# B&R Automation Studio project TD52 (part 51)

#### c_clutch_CANCyclic.st - Init, cyclic, exit code
```iecst
(*******************************************************************************
NOxSensor: 	 		CAN communication to Horton CAN bus device (cyclic)

This code is confidential and proprietary to the INNIO Company.
It may not be used in any form, or reproduced in any manner, without the express
written permission of the INNIO Company.
Copyright, INNIO Company, 2026

Customized modifications: -
------------------------

History:
-------

V4.16.00.00	06.01.2026	Bencze,  HORTON CAN bus device Cyclic code

Instructions for use:
--------------------

-----------------------------------------------------------------------------------------------------------------------------------------------	*)

PROGRAM _CYCLIC

	// Trigger reception of the data
	TON_1sTick(IN := NOT TON_1sTick.Q, PT := T#800ms);				(* 80ms + 2 times cycle time = 100ms *)

	// CAN communication timeout warning timers
	FOR DeviceNumber := 0 TO 3 DO
		TON_10sTick_DumpRadiator[DeviceNumber](IN := NOT DumpRadiator_PGN_Message_CS1[DeviceNumber].CommandDone OR NOT DumpRadiator_PGN_Message_CS2[DeviceNumber].CommandDone, PT := T#9800ms);
		TON_10sTick_AirInFan[DeviceNumber](IN := NOT AirInFan_PGN_Message_CS1[DeviceNumber].CommandDone OR NOT AirInFan_PGN_Message_CS2[DeviceNumber].CommandDone, PT := T#9800ms);
	END_FOR;

	// DumpRadiator - Connection with Map Services
	DumpRadiator_PGN_Message_CS1[0].MpLink := ADR(Dump_Radiator_1_CS1);
	DumpRadiator_PGN_Message_CS2[0].MpLink := ADR(Dump_Radiator_1_CS2);
	DumpRadiator_PGN_Message_CS1[1].MpLink := ADR(Dump_Radiator_2_CS1);
	DumpRadiator_PGN_Message_CS2[1].MpLink := ADR(Dump_Radiator_2_CS2);
	DumpRadiator_PGN_Message_CS1[2].MpLink := ADR(Dump_Radiator_3_CS1);
	DumpRadiator_PGN_Message_CS2[2].MpLink := ADR(Dump_Radiator_3_CS2);
	DumpRadiator_PGN_Message_CS1[3].MpLink := ADR(Dump_Radiator_4_CS1);
	DumpRadiator_PGN_Message_CS2[3].MpLink := ADR(Dump_Radiator_4_CS2);

	// AirInFan - Connection with Map Services
	AirInFan_PGN_Message_CS1[0].MpLink := ADR(Air_Inlet_Fan_1_CS1);
	AirInFan_PGN_Message_CS2[0].MpLink := ADR(Air_Inlet_Fan_1_CS2);
	AirInFan_PGN_Message_CS1[1].MpLink := ADR(Air_Inlet_Fan_2_CS1);
	AirInFan_PGN_Message_CS2[1].MpLink := ADR(Air_Inlet_Fan_2_CS2);
	AirInFan_PGN_Message_CS1[2].MpLink := ADR(Air_Inlet_Fan_3_CS1);
	AirInFan_PGN_Message_CS2[2].MpLink := ADR(Air_Inlet_Fan_3_CS2);
	AirInFan_PGN_Message_CS1[3].MpLink := ADR(Air_Inlet_Fan_4_CS1);
	AirInFan_PGN_Message_CS2[3].MpLink := ADR(Air_Inlet_Fan_4_CS2);

	FOR DeviceNumber := 0 TO 3 DO
		// Specific messages 1 (CS1 - Horton documentation)
		DumpRadiator_PGN_Message_CS1[DeviceNumber].Enable := TRUE;
		DumpRadiator_PGN_Message_CS1[DeviceNumber].Receive := TON_1sTick.Q;
		DumpRadiator_PGN_Message_CS1[DeviceNumber].PGN := 65470;
		DumpRadiator_PGN_Message_CS1[DeviceNumber].Priority := 5;
		DumpRadiator_PGN_Message_CS1[DeviceNumber].DataLength := 8;
		DumpRadiator_PGN_Message_CS1[DeviceNumber].Data := ADR(DumpRadiator_CS1_RawData[DeviceNumber]);
		DumpRadiator_PGN_Message_CS1[DeviceNumber]();

		// Specific messages 2 (CS2 - Horton documentation)
		DumpRadiator_PGN_Message_CS2[DeviceNumber].Enable := TRUE;
		DumpRadiator_PGN_Message_CS2[DeviceNumber].Receive := TON_1sTick.Q;
		DumpRadiator_PGN_Message_CS2[DeviceNumber].PGN := 65469;
		DumpRadiator_PGN_Message_CS2[DeviceNumber].Priority := 5;
		DumpRadiator_PGN_Message_CS2[DeviceNumber].DataLength := 8;
		DumpRadiator_PGN_Message_CS2[DeviceNumber].Data := ADR(DumpRadiator_CS2_RawData[DeviceNumber]);
		DumpRadiator_PGN_Message_CS2[DeviceNumber]();

		// Specific messages 1 (CS1 - Horton documentation)
		AirInFan_PGN_Message_CS1[DeviceNumber].Enable := TRUE;
		AirInFan_PGN_Message_CS1[DeviceNumber].Receive := TON_1sTick.Q;
		AirInFan_PGN_Message_CS1[DeviceNumber].PGN := 65470;
		AirInFan_PGN_Message_CS1[DeviceNumber].Priority := 5;
		AirInFan_PGN_Message_CS1[DeviceNumber].DataLength := 8;
		AirInFan_PGN_Message_CS1[DeviceNumber].Data := ADR(AirInFan_CS1_RawData[DeviceNumber]);
		AirInFan_PGN_Message_CS1[DeviceNumber]();

		// Specific messages 2 (CS2 - Horton documentation)
		AirInFan_PGN_Message_CS2[DeviceNumber].Enable := TRUE;
		AirInFan_PGN_Message_CS2[DeviceNumber].Receive := TON_1sTick.Q;
		AirInFan_PGN_Message_CS2[DeviceNumber].PGN := 65469;
		AirInFan_PGN_Message_CS2[DeviceNumber].Priority := 5;
		AirInFan_PGN_Message_CS2[DeviceNumber].DataLength := 8;
		AirInFan_PGN_Message_CS2[DeviceNumber].Data := ADR(AirInFan_CS2_RawData[DeviceNumber]);
		AirInFan_PGN_Message_CS2[DeviceNumber]();
	END_FOR;

	FOR DeviceNumber := 0 TO 3 DO
		// DumpRadiator - Measured Fan Speed and Speed signal from PLC (AO)
		MM2VIS_ThisPlant.rDumpRadiator_Speed[DeviceNumber] := DumpRadiator_CS1_RawData[DeviceNumber].Data2 + DumpRadiator_CS1_RawData[DeviceNumber].Data3 * 256; // Fan speed to the device
		MM2VIS_ThisPlant.rDumpRadiator_InputSpeed[DeviceNumber] := DumpRadiator_CS1_RawData[DeviceNumber].Data6 + DumpRadiator_CS1_RawData[DeviceNumber].Data7 * 256; // Fan speed measurement coming to PLC

		// AirInFan - Measured Fan Speed and Speed signal from PLC (AO)
		MM2VIS_ThisPlant.rAirInFan_Speed[DeviceNumber] := AirInFan_CS1_RawData[DeviceNumber].Data2 + AirInFan_CS1_RawData[DeviceNumber].Data3 * 256; // Fan speed to the device
		MM2VIS_ThisPlant.rAirInFan_InputSpeed[DeviceNumber]  := AirInFan_CS1_RawData[DeviceNumber].Data6 + AirInFan_CS1_RawData[DeviceNumber].Data7 * 256; // Fan speed measurement coming to PLC
	END_FOR;

	// Dump Radiators are running
	MM2VIS_ThisPlant.bDumpRadiatorRUN[0] := (MM2VIS_ThisPlant.rDumpRadiator_InputSpeed[0] >= OUT_CU.rCust_SparePara[26]);
	MM2VIS_ThisPlant.bDumpRadiatorRUN[1] := (MM2VIS_ThisPlant.rDumpRadiator_InputSpeed[1] >= OUT_CU.rCust_SparePara[26]);
	MM2VIS_ThisPlant.bDumpRadiatorRUN[2] := (MM2VIS_ThisPlant.rDumpRadiator_InputSpeed[2] >= OUT_CU.rCust_SparePara[26]);
	MM2VIS_ThisPlant.bDumpRadiatorRUN[3] := (MM2VIS_ThisPlant.rDumpRadiator_InputSpeed[3] >= OUT_CU.rCust_SparePara[26]);
	// Air Inlet Fans are running
	MM2VIS_ThisPlant.bAirInFanRUN[0] := (MM2VIS_ThisPlant.rAirInFan_InputSpeed[0] >= OUT_CU.rCust_SparePara[39]);
	MM2VIS_ThisPlant.bAirInFanRUN[1] := (MM2VIS_ThisPlant.rAirInFan_InputSpeed[1] >= OUT_CU.rCust_SparePara[39]);
	MM2VIS_ThisPlant.bAirInFanRUN[2] := (MM2VIS_ThisPlant.rAirInFan_InputSpeed[2] >= OUT_CU.rCust_SparePara[39]);
	MM2VIS_ThisPlant.bAirInFanRUN[3] := (MM2VIS_ThisPlant.rAirInFan_InputSpeed[3] >= OUT_CU.rCust_SparePara[39]);

	FOR DeviceNumber := 0 TO 3 DO
		// DumpRadiator - Clutch status
		MM2VIS_ThisPlant.bDumpRadiator_FanCmdLThanMICS[DeviceNumber] := DumpRadiator_CS2_RawData[DeviceNumber].Data2.3; // Fan command less than MICS (Min Controllable Fan Speed)
		MM2VIS_ThisPlant.bDumpRadiator_FanCmdLThanMITS[DeviceNumber] := DumpRadiator_CS2_RawData[DeviceNumber].Data2.4; // Fan command less than MITS (Min Maintained Fan Speed)
		MM2VIS_ThisPlant.bDumpRadiator_FanCmdGThanMax[DeviceNumber] := DumpRadiator_CS2_RawData[DeviceNumber].Data2.5; // Fan command greater than Max Fan Speed.
		MM2VIS_ThisPlant.bDumpRadiator_InputSpeedGThanM[DeviceNumber] := DumpRadiator_CS2_RawData[DeviceNumber].Data2.6; // Input speed greater than MAOS (Max Allowed Operating Fan Speed)

		MM2VIS_ThisPlant.bDumpRadiator_SPN2978InputFault[DeviceNumber] := DumpRadiator_CS2_RawData[DeviceNumber].Data4.0; // SPN2978 Input Fault
		MM2VIS_ThisPlant.bDumpRadiator_FanSpeedPinFault[DeviceNumber] := DumpRadiator_CS2_RawData[DeviceNumber].Data4.1; // Fan Speed Pin Fault
		MM2VIS_ThisPlant.bDumpRadiator_NoFanSpeed[DeviceNumber] := DumpRadiator_CS2_RawData[DeviceNumber].Data4.2; // No Fan Speed
		MM2VIS_ThisPlant.bDumpRadiator_ExcessFanSpeed[DeviceNumber] := DumpRadiator_CS2_RawData[DeviceNumber].Data4.3; // Excess Fan Speed
		MM2VIS_ThisPlant.bDumpRadiator_FanSpeedError[DeviceNumber] := DumpRadiator_CS2_RawData[DeviceNumber].Data4.4; // Fan Speed Error
		MM2VIS_ThisPlant.bDumpRadiator_OutputHWFault[DeviceNumber] := DumpRadiator_CS2_RawData[DeviceNumber].Data4.5; // Output Hardware Fault (MUST REPLACE CONTROLLER)
		MM2VIS_ThisPlant.bDumpRadiator_APTFault[DeviceNumber] := DumpRadiator_CS2_RawData[DeviceNumber].Data4.6; // APT Fault
		MM2VIS_ThisPlant.bDumpRadiator_InputSpeedError[DeviceNumber] := DumpRadiator_CS2_RawData[DeviceNumber].Data4.7; // Input Speed Error

		MM2VIS_ThisPlant.bDumpRadiator_APPFault[DeviceNumber] := DumpRadiator_CS2_RawData[DeviceNumber].Data5.3; // APP Fault
		MM2VIS_ThisPlant.bDumpRadiator_EngineRPMFault[DeviceNumber] := DumpRadiator_CS2_RawData[DeviceNumber].Data5.4; // Engine RPM Fault
		MM2VIS_ThisPlant.bDumpRadiator_ClutchOutputShort[DeviceNumber] := DumpRadiator_CS2_RawData[DeviceNumber].Data5.5; // Fan Clutch Output Short
		MM2VIS_ThisPlant.bDumpRadiator_ClutchOutputOpen[DeviceNumber] := DumpRadiator_CS2_RawData[DeviceNumber].Data5.6; // Fan Clutch Output Open
		MM2VIS_ThisPlant.bDumpRadiator_ClutchOutputFault[DeviceNumber] := DumpRadiator_CS2_RawData[DeviceNumber].Data5.7; // Fan Clutch Output Fault
		MM2VIS_ThisPlant.bDumpRadiator_InputPowerLow[DeviceNumber] := DumpRadiator_CS2_RawData[DeviceNumber].Data6.0; // Input Power Low
		MM2VIS_ThisPlant.bDumpRadiator_InputPowerHigh[DeviceNumber] := DumpRadiator_CS2_RawData[DeviceNumber].Data6.1; // Input Power High
		MM2VIS_ThisPlant.bDumpRadiator_InputPowerFault[DeviceNumber] := DumpRadiator_CS2_RawData[DeviceNumber].Data6.2; // Input Power Fault
		MM2VIS_ThisPlant.bDumpRadiator_SensorPowerLow[DeviceNumber] := DumpRadiator_CS2_RawData[DeviceNumber].Data6.3; // Sensor Power Low
		MM2VIS_ThisPlant.bDumpRadiator_SensorPowerHigh[DeviceNumber] := DumpRadiator_CS2_RawData[DeviceNumber].Data6.4; // Sensor Power High
		MM2VIS_ThisPlant.bDumpRadiator_SensorPowerFault[DeviceNumber] := DumpRadiator_CS2_RawData[DeviceNumber].Data6.5; // Sensor Power Fault
		MM2VIS_ThisPlant.bDumpRadiator_EngSpeedLow[DeviceNumber] := DumpRadiator_CS2_RawData[DeviceNumber].Data6.6; // Engagement fault (fan speed low)
		MM2VIS_ThisPlant.bDumpRadiator_DisEngSpeedHigh[DeviceNumber] := DumpRadiator_CS2_RawData[DeviceNumber].Data6.7; // Disengagement fault (fan speed high)

		// DumpRadiator - Warning messages - Status
		MM2VIS_ThisPlant.bDumpRadiator_WarningMsg[DeviceNumber] := 	MM2VIS_ThisPlant.bDumpRadiator_FanCmdLThanMICS[DeviceNumber]	OR MM2VIS_ThisPlant.bDumpRadiator_FanCmdLThanMITS[DeviceNumber] 	OR
		MM2VIS_ThisPlant.bDumpRadiator_FanCmdGThanMax[DeviceNumber] 	OR MM2VIS_ThisPlant.bDumpRadiator_InputSpeedGThanM[DeviceNumber] 	OR
		MM2VIS_ThisPlant.bDumpRadiator_SPN2978InputFault[DeviceNumber] 	OR MM2VIS_ThisPlant.bDumpRadiator_FanSpeedPinFault[DeviceNumber] 	OR
		MM2VIS_ThisPlant.bDumpRadiator_NoFanSpeed[DeviceNumber] 		OR MM2VIS_ThisPlant.bDumpRadiator_ExcessFanSpeed[DeviceNumber] 		OR
		MM2VIS_ThisPlant.bDumpRadiator_FanSpeedError[DeviceNumber] 		OR MM2VIS_ThisPlant.bDumpRadiator_OutputHWFault[DeviceNumber] 		OR
		MM2VIS_ThisPlant.bDumpRadiator_APTFault[DeviceNumber] 			OR MM2VIS_ThisPlant.bDumpRadiator_InputSpeedError[DeviceNumber] 	OR
		MM2VIS_ThisPlant.bDumpRadiator_APPFault[DeviceNumber] 			OR MM2VIS_ThisPlant.bDumpRadiator_EngineRPMFault[DeviceNumber] 		OR
		MM2VIS_ThisPlant.bDumpRadiator_ClutchOutputShort[DeviceNumber] 	OR MM2VIS_ThisPlant.bDumpRadiator_ClutchOutputOpen[DeviceNumber] 	OR
		MM2VIS_ThisPlant.bDumpRadiator_ClutchOutputFault[DeviceNumber] 	OR MM2VIS_ThisPlant.bDumpRadiator_InputPowerLow[DeviceNumber] 		OR
		MM2VIS_ThisPlant.bDumpRadiator_InputPowerHigh[DeviceNumber] 	OR MM2VIS_ThisPlant.bDumpRadiator_InputPowerFault[DeviceNumber] 	OR
		MM2VIS_ThisPlant.bDumpRadiator_SensorPowerLow[DeviceNumber] 	OR MM2VIS_ThisPlant.bDumpRadiator_SensorPowerHigh[DeviceNumber] 	OR
		MM2VIS_ThisPlant.bDumpRadiator_SensorPowerFault[DeviceNumber] 	OR MM2VIS_ThisPlant.bDumpRadiator_EngSpeedLow[DeviceNumber] 		OR
		MM2VIS_ThisPlant.bDumpRadiator_DisEngSpeedHigh[DeviceNumber];

		// AirInFan - Clutch status
		MM2VIS_ThisPlant.bAirInFan_FanCmdLThanMICS[DeviceNumber] := AirInFan_CS2_RawData[DeviceNumber].Data2.3; // Fan command less than MICS (Min Controllable Fan Speed)
		MM2VIS_ThisPlant.bAirInFan_FanCmdLThanMITS[DeviceNumber] := AirInFan_CS2_RawData[DeviceNumber].Data2.4; // Fan command less than MITS (Min Maintained Fan Speed)
		MM2VIS_ThisPlant.bAirInFan_FanCmdGThanMax[DeviceNumber] := AirInFan_CS2_RawData[DeviceNumber].Data2.5; // Fan command greater than Max Fan Speed.
		MM2VIS_ThisPlant.bAirInFan_InputSpeedGThanM[DeviceNumber] := AirInFan_CS2_RawData[DeviceNumber].Data2.6; // Input speed greater than MAOS (Max Allowed Operating Fan Speed)

		MM2VIS_ThisPlant.bAirInFan_SPN2978InputFault[DeviceNumber] := AirInFan_CS2_RawData[DeviceNumber].Data4.0; // SPN2978 Input Fault
		MM2VIS_ThisPlant.bAirInFan_FanSpeedPinFault[DeviceNumber] := AirInFan_CS2_RawData[DeviceNumber].Data4.1; // Fan Speed Pin Fault
		MM2VIS_ThisPlant.bAirInFan_NoFanSpeed[DeviceNumber] := AirInFan_CS2_RawData[DeviceNumber].Data4.2; // No Fan Speed
		MM2VIS_ThisPlant.bAirInFan_ExcessFanSpeed[DeviceNumber] := AirInFan_CS2_RawData[DeviceNumber].Data4.3; // Excess Fan Speed
		MM2VIS_ThisPlant.bAirInFan_FanSpeedError[DeviceNumber] := AirInFan_CS2_RawData[DeviceNumber].Data4.4; // Fan Speed Error
		MM2VIS_ThisPlant.bAirInFan_OutputHWFault[DeviceNumber] := AirInFan_CS2_RawData[DeviceNumber].Data4.5; // Output Hardware Fault (MUST REPLACE CONTROLLER)
		MM2VIS_ThisPlant.bAirInFan_APTFault[DeviceNumber] := AirInFan_CS2_RawData[DeviceNumber].Data4.6; // APT Fault
		MM2VIS_ThisPlant.bAirInFan_InputSpeedError[DeviceNumber] := AirInFan_CS2_RawData[DeviceNumber].Data4.7; // Input Speed Error

		MM2VIS_ThisPlant.bAirInFan_APPFault[DeviceNumber] := AirInFan_CS2_RawData[DeviceNumber].Data5.3; // APP Fault
		MM2VIS_ThisPlant.bAirInFan_EngineRPMFault[DeviceNumber] := AirInFan_CS2_RawData[DeviceNumber].Data5.4; // Engine RPM Fault
		MM2VIS_ThisPlant.bAirInFan_ClutchOutputShort[DeviceNumber] := AirInFan_CS2_RawData[DeviceNumber].Data5.5; // Fan Clutch Output Short
		MM2VIS_ThisPlant.bAirInFan_ClutchOutputOpen[DeviceNumber] := AirInFan_CS2_RawData[DeviceNumber].Data5.6; // Fan Clutch Output Open
		MM2VIS_ThisPlant.bAirInFan_ClutchOutputFault[DeviceNumber] := AirInFan_CS2_RawData[DeviceNumber].Data5.7; // Fan Clutch Output Fault
		MM2VIS_ThisPlant.bAirInFan_InputPowerLow[DeviceNumber] := AirInFan_CS2_RawData[DeviceNumber].Data6.0; // Input Power Low
		MM2VIS_ThisPlant.bAirInFan_InputPowerHigh[DeviceNumber] := AirInFan_CS2_RawData[DeviceNumber].Data6.1; // Input Power High
		MM2VIS_ThisPlant.bAirInFan_InputPowerFault[DeviceNumber] := AirInFan_CS2_RawData[DeviceNumber].Data6.2; // Input Power Fault
		MM2VIS_ThisPlant.bAirInFan_SensorPowerLow[DeviceNumber] := AirInFan_CS2_RawData[DeviceNumber].Data6.3; // Sensor Power Low
		MM2VIS_ThisPlant.bAirInFan_SensorPowerHigh[DeviceNumber] := AirInFan_CS2_RawData[DeviceNumber].Data6.4; // Sensor Power High
		MM2VIS_ThisPlant.bAirInFan_SensorPowerFault[DeviceNumber] := AirInFan_CS2_RawData[DeviceNumber].Data6.5; // Sensor Power Fault
		MM2VIS_ThisPlant.bAirInFan_EngSpeedLow[DeviceNumber] := AirInFan_CS2_RawData[DeviceNumber].Data6.6; // Engagement fault (fan speed low)
		MM2VIS_ThisPlant.bAirInFan_DisEngSpeedHigh[DeviceNumber] := AirInFan_CS2_RawData[DeviceNumber].Data6.7; // Disengagement fault (fan speed high)

		// AirInFan - Warning messages - Status
		MM2VIS_ThisPlant.bAirInFan_WarningMsg[DeviceNumber] := 	MM2VIS_ThisPlant.bAirInFan_FanCmdLThanMICS[DeviceNumber]	OR MM2VIS_ThisPlant.bAirInFan_FanCmdLThanMITS[DeviceNumber] 	OR
		MM2VIS_ThisPlant.bAirInFan_FanCmdGThanMax[DeviceNumber] 	OR MM2VIS_ThisPlant.bAirInFan_InputSpeedGThanM[DeviceNumber] 	OR
		MM2VIS_ThisPlant.bAirInFan_SPN2978InputFault[DeviceNumber] 	OR MM2VIS_ThisPlant.bAirInFan_FanSpeedPinFault[DeviceNumber]	OR
		MM2VIS_ThisPlant.bAirInFan_NoFanSpeed[DeviceNumber] 		OR MM2VIS_ThisPlant.bAirInFan_ExcessFanSpeed[DeviceNumber]		OR
		MM2VIS_ThisPlant.bAirInFan_FanSpeedError[DeviceNumber] 		OR MM2VIS_ThisPlant.bAirInFan_OutputHWFault[DeviceNumber] OR
		MM2VIS_ThisPlant.bAirInFan_APTFault[DeviceNumber] 			OR MM2VIS_ThisPlant.bAirInFan_InputSpeedError[DeviceNumber] 	OR
		MM2VIS_ThisPlant.bAirInFan_APPFault[DeviceNumber] 			OR MM2VIS_ThisPlant.bAirInFan_EngineRPMFault[DeviceNumber] 		OR
		MM2VIS_ThisPlant.bAirInFan_ClutchOutputShort[DeviceNumber] 	OR MM2VIS_ThisPlant.bAirInFan_ClutchOutputOpen[DeviceNumber] 	OR
		MM2VIS_ThisPlant.bAirInFan_ClutchOutputFault[DeviceNumber] 	OR MM2VIS_ThisPlant.bAirInFan_InputPowerLow[DeviceNumber] 		OR
		MM2VIS_ThisPlant.bAirInFan_InputPowerHigh[DeviceNumber]		OR MM2VIS_ThisPlant.bAirInFan_InputPowerFault[DeviceNumber] 	OR
		MM2VIS_ThisPlant.bAirInFan_SensorPowerLow[DeviceNumber] 	OR MM2VIS_ThisPlant.bAirInFan_SensorPowerHigh[DeviceNumber] 	OR
		MM2VIS_ThisPlant.bAirInFan_SensorPowerFault[DeviceNumber]	OR MM2VIS_ThisPlant.bAirInFan_EngSpeedLow[DeviceNumber] 		OR
		MM2VIS_ThisPlant.bAirInFan_DisEngSpeedHigh[DeviceNumber];
	END_FOR;

	// CAN error - Reset the data
	FOR DeviceNumber := 0 TO 3 DO
		IF TON_10sTick_DumpRadiator[DeviceNumber].Q THEN
			DumpRadiator_CS1_RawData[DeviceNumber].Data0 := 0;
			DumpRadiator_CS1_RawData[DeviceNumber].Data1 := 0;
			DumpRadiator_CS1_RawData[DeviceNumber].Data2 := 0;
			DumpRadiator_CS1_RawData[DeviceNumber].Data3 := 0;
			DumpRadiator_CS1_RawData[DeviceNumber].Data4 := 0;
			DumpRadiator_CS1_RawData[DeviceNumber].Data5 := 0;
			DumpRadiator_CS1_RawData[DeviceNumber].Data6 := 0;
			DumpRadiator_CS1_RawData[DeviceNumber].Data7 := 0;

			DumpRadiator_CS2_RawData[DeviceNumber].Data0 := 0;
			DumpRadiator_CS2_RawData[DeviceNumber].Data1 := 0;
			DumpRadiator_CS2_RawData[DeviceNumber].Data2 := 0;
			DumpRadiator_CS2_RawData[DeviceNumber].Data3 := 0;
			DumpRadiator_CS2_RawData[DeviceNumber].Data4 := 0;
			DumpRadiator_CS2_RawData[DeviceNumber].Data5 := 0;
			DumpRadiator_CS2_RawData[DeviceNumber].Data6 := 0;
			DumpRadiator_CS2_RawData[DeviceNumber].Data7 := 0;
		END_IF;

		IF TON_10sTick_AirInFan[DeviceNumber].Q THEN
			AirInFan_CS1_RawData[DeviceNumber].Data0 := 0;
			AirInFan_CS1_RawData[DeviceNumber].Data1 := 0;
			AirInFan_CS1_RawData[DeviceNumber].Data2 := 0;
			AirInFan_CS1_RawData[DeviceNumber].Data3 := 0;
			AirInFan_CS1_RawData[DeviceNumber].Data4 := 0;
			AirInFan_CS1_RawData[DeviceNumber].Data5 := 0;
			AirInFan_CS1_RawData[DeviceNumber].Data6 := 0;
			AirInFan_CS1_RawData[DeviceNumber].Data7 := 0;

			AirInFan_CS2_RawData[DeviceNumber].Data0 := 0;
			AirInFan_CS2_RawData[DeviceNumber].Data1 := 0;
			AirInFan_CS2_RawData[DeviceNumber].Data2 := 0;
			AirInFan_CS2_RawData[DeviceNumber].Data3 := 0;
			AirInFan_CS2_RawData[DeviceNumber].Data4 := 0;
			AirInFan_CS2_RawData[DeviceNumber].Data5 := 0;
			AirInFan_CS2_RawData[DeviceNumber].Data6 := 0;
			AirInFan_CS2_RawData[DeviceNumber].Data7 := 0;
		END_IF;
	END_FOR;

	// CAN status to VISU
	FOR DeviceNumber := 0 TO 3 DO
		MM2VIS_ThisPlant.bDumpRadiatorCAN[DeviceNumber] := TON_10sTick_DumpRadiator[DeviceNumber].Q;
		MM2VIS_ThisPlant.bAirInFanCAN[DeviceNumber] := TON_10sTick_AirInFan[DeviceNumber].Q;
	END_FOR;

	// CAN Warning messages
	MM2VIS_ThisPlant.bDumpRadiator_CANWarningMsg := 	MM2VIS_ThisPlant.bDumpRadiatorCAN[0] OR MM2VIS_ThisPlant.bDumpRadiatorCAN[1] OR
	MM2VIS_ThisPlant.bDumpRadiatorCAN[2] OR MM2VIS_ThisPlant.bDumpRadiatorCAN[3];

	MM2VIS_ThisPlant.bAirInFan_CANWarningMsg := 	MM2VIS_ThisPlant.bAirInFanCAN[0] OR MM2VIS_ThisPlant.bAirInFanCAN[1] OR
	MM2VIS_ThisPlant.bAirInFanCAN[2] OR MM2VIS_ThisPlant.bAirInFanCAN[3];

END_PROGRAM
```

#### c_clutch_CAN.var - Local variables
```iecst
VAR
	AirInFan_CS2_RawData : ARRAY[0..3] OF CS2_Data;
	AirInFan_CS1_RawData : ARRAY[0..3] OF CS1_Data;
	DumpRadiator_CS2_RawData : ARRAY[0..3] OF CS2_Data;
	DumpRadiator_CS1_RawData : ARRAY[0..3] OF CS1_Data;
	AirInFan_PGN_Message_CS1 : ARRAY[0..3] OF MpJ1939Receive;
	AirInFan_PGN_Message_CS2 : ARRAY[0..3] OF MpJ1939Receive;
	DumpRadiator_PGN_Message_CS1 : ARRAY[0..3] OF MpJ1939Receive;
	DumpRadiator_PGN_Message_CS2 : ARRAY[0..3] OF MpJ1939Receive;
	TON_10sTick_AirInFan : ARRAY[0..3] OF TON;
	TON_10sTick_DumpRadiator : ARRAY[0..3] OF TON;
	TON_1sTick : TON;
	DeviceNumber : INT := 0;
END_VAR
```

#### c_clutch_CAN.typ - Local data types
```iecst
TYPE
	CS2_Data : 	STRUCT
		Data0 : USINT;
		Data1 : USINT;
		Data2 : USINT;
		Data3 : USINT;
		Data4 : USINT;
		Data5 : USINT;
		Data6 : USINT;
		Data7 : USINT;
	END_STRUCT;
	CS1_Data : 	STRUCT
		Data0 : USINT;
		Data1 : USINT;
		Data2 : USINT;
		Data3 : USINT;
		Data4 : USINT;
		Data5 : USINT;
		Data6 : USINT;
		Data7 : USINT;
	END_STRUCT;
END_TYPE
```

### Package Logical/Emission - EM: Emission Control

### Package Logical/Emission/Lib_EM - Libraries

### Library Logical/Emission/Lib_EM/lUDC (ANSIC)

#### lUDC.fun
```iecst
FUNCTION_BLOCK fUDC
  VAR_INPUT
    ssMethodType: SINT;
  END_VAR  VAR_INPUT
        Para : tUD_PARA; (**)
  END_VAR
  VAR_INPUT
        In : tUD_IN; (**)
  END_VAR
  VAR_INPUT
        Perm : tUD_PERM; (**)
  END_VAR
 VAR_OUTPUT
        dbg : tUD_DBG; (**)
  END_VAR
 VAR_OUTPUT
        Out : tUD_OUT; (**)
  END_VAR
  VAR_OUTPUT
        Version : UDINT; (**)
  END_VAR
	VAR
		bur_BlockIO_UDC : BlockIO_UDC;
	END_VAR
	VAR
		bur_D_Work_UDC : D_Work_UDC;
	END_VAR
	VAR
		bur_ExternalInputs_UDC : ExternalInputs_UDC;
	END_VAR
	VAR
		bur_ExternalOutputs_UDC : ExternalOutputs_UDC;
	END_VAR
	VAR
		bur_UDC : tag_RTM_UDC;
	END_VAR
END_FUNCTION_BLOCK
```

#### lUDC.typ
```iecst
TYPE

   tHALioAi : STRUCT
        Ai : REAL; (* ()*)
        Unfilt : REAL; (* ()*)
        GoodQual : BOOL; (* ()*)
    END_STRUCT;

   tUD_CLFlow_DBG : STRUCT
        up : REAL; (*proportional part ()*)
        ui : REAL; (*integral part ()*)
        ud : REAL; (*derivative part ()*)
        aw : REAL; (*anti windup ()*)
    END_STRUCT;

   tUD_CLNOx_DBG : STRUCT
        up : REAL; (*proportional part ()*)
        ui : REAL; (*integral part ()*)
        ud : REAL; (*derivative part ()*)
        aw : REAL; (*anti windup ()*)
        bFreeze : BOOL; (*Freeze controller ()*)
        bSatUpLim : BOOL; (*Controller saturated at upper limit ()*)
    END_STRUCT;

   tUD_CLNOx_PERM : STRUCT
        rUrClKawExt : REAL; (*Anti windup gain for external output limitation  of closed loop urea injection controller (ppm*h/l)*)
        rUrClKaw : REAL; (*Anti windup gain for internal output limitation  of closed loop urea injection controller (ppm*h/l)*)
        rUrClN : REAL; (*Derivative filter bandwith of PID closed loop urea injection controller offset (1/s)*)
        rUrClKdOffs_x : ARRAY[0..4] OF REAL; (*Derivative gain of PID closed loop urea injection controller offset (degC)*)
        rUrClKdOffs_y : ARRAY[0..4] OF REAL; (*Derivative gain of PID closed loop urea injection controller offset (l*s/(h*ppm))*)
        rUrClKiOffs_x : ARRAY[0..4] OF REAL; (*Integral gain of PID closed loop urea injection controller offset (degC)*)
        rUrClKiOffs_y : ARRAY[0..4] OF REAL; (*Integral gain of PID closed loop urea injection controller offset (l/(h*ppm*s))*)
        rUrClKpOffs_x : ARRAY[0..4] OF REAL; (*proportional gain of PID closed loop urea injection controller offset (degC)*)
        rUrClKpOffs_y : ARRAY[0..4] OF REAL; (*proportional gain of PID closed loop urea injection controller offset (l/(h*ppm))*)
        rUrClD0 : REAL; (*If PID closed loop urea flow controller is reseted, its derivate filter output is reseted to this value (-)*)
        rUrClI0 : REAL; (*If PID closed loop urea flow controller is reseted, its integral output is reseted to this value (l/h)*)
        bUrClRes : BOOL; (*If TRUE,  resets the PID closed loop urea flow controller to reset value. (-)*)
    END_STRUCT;

   tUD_CLPp_PERM : STRUCT
        rUrPpKawExt : REAL; (*External anti windup gain for urea injection control via urea pump speed (tbd)*)
        rUrPpKaw : REAL; (*Internal anti windup gain for urea injection control via urea pump speed (tbd)*)
        rUrPpN : REAL; (*1st order filter frequency for derivative gain  of pump speed based urea injection controller (PIDN) (tbd)*)
        rUrPpKdOffs : REAL; (*Derivative gain  of pump speed based urea injection controller offset (PIDN) (tbd)*)
        rUrPpKiOffs : REAL; (*Integral gain  of pump speed based urea injection controller offset (PIDN) (tbd)*)
        rUrPpKpOffs : REAL; (*Proportional gain  of pump speed based urea injection controller offset (PIDN) (tbd)*)
        rUrPpD0 : REAL; (*Initial value for derviative 1st order filter  of pump speed based urea injection controller (PIDN) (tbd)*)
        rUrPpI0 : REAL; (*Initial value for integrator of pump speed based urea injection controller (PIDN) (tbd)*)
        bUrPpRes : BOOL; (*Reset for pump speed based urea injection controller,  reset if = TRUE (-)*)
        rUrPpCntrFFMap_x : ARRAY[0..10] OF REAL; (*tbd (l/h)*)
        rUrPpCntrFFMap_y : ARRAY[0..10] OF REAL; (*tbd (au)*)
    END_STRUCT;

   tUD_CLVal_PERM : STRUCT
        rUrValKawExt : REAL; (*External anti windup gain for urea valve closed loop controller (tbd)*)
        rUrValKaw : REAL; (*Internal anti windup gain for urea valve closed loop controller (tbd)*)
        rUrValN : REAL; (*Filter frequency constant of PIDN based urea valve closed loop controller (tbd)*)
        rUrValKdOffs : REAL; (*Derivative gain of PIDN based urea valve closed loop controller offset (tbd)*)
        rUrValKiOffs : REAL; (*Integral gain of PIDN based urea valve closed loop controller offset (tbd)*)
        rUrValKpOffs : REAL; (*Proportional gain of PIDN based urea valve closed loop controller offset (tbd)*)
        rUrValD0 : REAL; (*Initial value for derivative filter of PIDN based urea valve closed loop controller (tbd)*)
        rUrValI0 : REAL; (*Initial condition of integrator of PIDN based urea valve closed loop controller (au)*)
        bUrValRes : BOOL; (*Reset for PIDN based urea valve closed loop controller. Reset if TRUE (-)*)
        rUrValLinMap_x : ARRAY[0..10] OF REAL; (*Linearisation curve for urea dosage valve input vector; Valve output, Kv/Kvs (au)*)
        rUrValLinMap_y : ARRAY[0..10] OF REAL; (*Linearisation curve for urea dosage valve output vector; Valve output, Reference value for urea dosage valve position (au)*)
        rTiFilt_DPrVlv : REAL; (*Filter time constant for the filtered differential pressure of the urea dosing valve (s)*)
    END_STRUCT;

   tUD_DBG : STRUCT
        SM : tUD_SM_DBG; (*Debug bus Signal Manager ()*)
        FF : tUD_FF_DBG; (*Debug bus Feed Forward ()*)
        Slip : tUD_Slip_DBG; (*Debug bus Slip Detection ()*)
        CLNOx : tUD_CLNOx_DBG; (*Debug bus Closed Loop ()*)
        CLFlow : tUD_CLFlow_DBG; (*Debug bus Closed Loop ()*)
    END_STRUCT;

   tUD_EMLine : STRUCT
        rCO : REAL; (* (ppm)*)
        rNO : REAL; (* (ppm)*)
        rNO2 : REAL; (* (ppm)*)
        bCO : BOOL; (* (-)*)
        bNO : BOOL; (* (-)*)
        bNO2 : BOOL; (* (-)*)
        bRdy : BOOL; (* (-)*)
    END_STRUCT;

   tUD_FF_DBG : STRUCT
        rSV : REAL; (*Space velocity through catalyst (1/h)*)
        rMdot_exh : REAL; (*Estimated exhaust mass flow [kg/s] (kg/s)*)
        rTSCRAvgEst : REAL; (*Estimated average SCR surface temperature (averaged over all cells) by observer (°C)*)
        rTSCRAvgAr : REAL; (*Arithmetic weighted average of SCR temperature using exhaust gas input and output temperature (°C)*)
        rTSCRAvg : REAL; (*Average SCR temperature used for NH3 feed forward control and urea injection start decision (°C)*)
        rNH3StDMaxAvgEst : REAL; (*Max NH3 storage capacity caluclated based on estimated average SCR temperature using temperature observer (g/m2)*)
        rNH3StDMaxAr : REAL; (*Max NH3 storage capacity calculated based on arithmetic weighted SCR temperature dervied from exhaust gas input and output temperature (g/m2)*)
        rNH3StDEst : REAL; (*Estimation of the actual NH3 storage density (mass of ammonia per m2 of active SCR surface) inside the SCR (g/m2)*)
        rNH3InFFSS : REAL; (*Ouput of the NH3 steady state feed forwward injection controller (ppm)*)
        rNH3InFF : REAL; (*Output of the feed forward NH3 injection controller (ppm)*)
        rdeltaNH3InTr : REAL; (*Ouput of the NH3 transient feed forward injection controller (ppm)*)
        rdeltaNH3InTr2 : REAL; (*Output of second transient feed forward controller based on Nox measurements ()*)
        rNH3StDEst2 : REAL; (*Actual NH3 storage estimated by second transient feed forward controller based on Nox measurements  ()*)
        iIdxFFOut : USINT; (*Urea injection feed forward idx ()*)
        rFlowUreaFF_LT : REAL; (*Urea injection FF load table dependend calculation (l/h)*)
        rFlowUreaFF_NOx : REAL; (*Urea injection FF engine  NOx based (l/h)*)
        rFlowUreaFF_Map : REAL; (*Urea injection FF map based (massflow, temp, NOx) (l/h)*)
        rFlowUreaFF_NH3 : REAL; (*Urea injection FF NH3 sensor based (l/h)*)
        rDensUrea : REAL; (*Urea density (g/l)*)
    END_STRUCT;

   tUD_FF_PERM : STRUCT
        rNH3FFMinLim : REAL; (*Minimum limit of output of ammonia feed forward controller (ppm)*)
        rNH3FFMaxLim : REAL; (*Maximum limit of output of ammonia feed forward controller (ppm)*)
        rdNH3TrMinLim : REAL; (*Minimum limit for transient feed forward NH3 injection control (ppm)*)
        rdNH3TrMaxLim : REAL; (*Maximum limit for transient feed forward NH3 injection control (ppm)*)
        rTSCRInit : REAL; (*Initial / reset value of SCR surface temperature output (degC)*)
        bTSCRRes : BOOL; (*If TRUE,  SCR surface temperature output is reset to I0 (initial temperature) (-)*)
        rNH3SSCor : REAL; (*Correction factor for steady state feedforward controller output (-)*)
        bNH3StDRes : BOOL; (*If TRUE resets the integrator of the estimated ammonia storage density (-)*)
        rNH3InTrGainB : REAL; (*Gain B for the transient feed forward NH3 injection controller. Increasing this value makes the transient FF term initially higher and reduction over time faster. (ppm*m2/g)*)
        rNH3InTrGainA : REAL; (*Gain A for the transient feed forward NH3 injection controller. Increasing this value fades out the transient feed forward term faster over time. (g/(m2*s*ppm))*)
        rMwUr : REAL; (*Mole weight of urea (g/mol)*)
        rMwExh : REAL; (*Mole weight of exhaust gas (g/mol)*)
        rUrFFMinLim : REAL; (*Minimum limitation of output of feed forward urea injection controller including adaptation of output via master controller gain plus offset (l/h)*)
        rUrFFMaxLim : REAL; (*Maximum limitation of output of feed forward urea injection controller including adaptation of output via master controller gain plus offset (l/h)*)
        bNH3InFFSSEn : BOOL; (*Enables steady state feed forward NH3 injection calculation if = TRUE According to spec doc D1-c (-)*)
        bdeltNH3InTrEn : BOOL; (*Enables transient feed forward NH3 injection calculation if = TRUE (-)*)
        bUrInModEn : BOOL; (*Enables model based feed forward urea injection calculation if = TRUE according to spec doc D1-d (-)*)
        rNH3StorMap_x : ARRAY[0..4] OF REAL; (*Estimated SCR temperature (degC)*)
        rNH3StorMap_y : ARRAY[0..4] OF REAL; (*Estimated max NH3 storage capacity (g/m2)*)
        bTSCRObsEn : BOOL; (*Activates the SCR temperature observer and uses Observer ouput to calculate average temeprature and max NH3 storage capacity, if = TRUE; Uses arithmetic mean to calculate SCR temperature and max storage capacity if = False (-)*)
        rNOxRedRatioMap_SV : ARRAY[0..2] OF REAL; (*Maximum NOx reduction ratio based on SCR temperature and exhaust space velocity SV: input SV (1/h)*)
        rNOxRedRatioMap_T : ARRAY[0..5] OF REAL; (*Maximum NOx reduction ratio based on SCR temperature and exhaust space velocity: input T (degC)*)
        rNOxRedRatioMap_out : ARRAY[0..17] OF REAL; (*Maximum NOx reduction ratio based on SCR temperature and exhaust space velocity: output (au)*)
        bdeltNH3InTrEn2 : BOOL; (*Release of second transient feed forward Urea controller output ()*)
        rNH3InTrGainC : REAL; (*Input gain of second transient feed forward Urea controller (g/m2/s/ppm)*)
        rNH3InTrGainD : REAL; (*Output gain of second transient feed forward Urea controller (ppm*m2/g)*)
        bNH3StDRes2 : BOOL; (*Reset of second transient feed forward Urea controller integrator ()*)
        rGainDeload : REAL; (*Deloading gain of second transient feed forward Urea controller (1/s)*)
        rdNH3TrMaxLim2 : REAL; (*Maximum output limit of second transient feed forward Urea controller (ppm)*)
        rdNH3TrMinLim2 : REAL; (*Maximum output limit of second transient feed forward Urea controller (ppm)*)
        rNH3SensStepUp : REAL; (*Upwards step of NH3 Sensor based urea injection closed loop controller (ppm)*)
        rNH3SensStepDwn : REAL; (*Downwards step of NH3 Sensor based urea injection closed loop controller (ppm)*)
        rNH3SensTrDel : REAL; (*Transport delay for NH3 Sensor based urea injection closed loop controller (s)*)
        rNH3SensGain : REAL; (*Proportional gain for NH3 Sensor based urea injection closed loop controller (-)*)
        bSCR_NH3Control_Active : BOOL; (*If TRUE, NH3 sensor based Urea injection closed loop control is enabled (-)*)
        rA_SCR_CatSurfaceOuter : REAL; (*Catalyst outer surface. Used for heat transfer calculations to the ambient (m2)*)
        rT_SCR_CatHeatTrans_Coef : REAL; (*Heat transfer coefficient from catalyst surface to ambient. Consider isolation material,  therefore assume very low values. (W/m2K)*)
        rC_SCR_ExhaustGas : REAL; (*Specific heat capacity of exhaust gas at constant pressure (J/kgK)*)
        rC_SCR_Cat : REAL; (*Specific heat capacity of catalyst material (mainly of the steel carrier material) (J/kgK)*)
        rMass_SCR_Cat : REAL; (*Mass of the catalyst (kg)*)
        rTmass_SCR_Cat : REAL; (*Thermal mass of catalyst housing (kJ/K)*)
        rNRho_SCR_WetExhaust : REAL; (*Density of the wet exhaust gas in kg per norm m3  P21 measurements for typical values: wet: 1.264 kg/Nm3 dry: 1.318 kg/Nm3 (kg/Nm3)*)
        rPnorm_Thresh : REAL; (*Power (normalized) threshold for activation of SCR feed forward adjustment (-)*)
        rTiConstAvgOn : REAL; (*Time constant after which the averaging of actual FF urea mass flow and the measured urea flow starts (s)*)
        rTiConstAvgOff : REAL; (*Time constant which determines the waiting period until the new averaging of actual FF urea mass flow and the measured urea flow starts (s)*)
        rTiFiltUreaFFAdjust : REAL; (*Time constant of the PT1 filter for the actual NH3 mass flow rate (s)*)
        rUreaGainDeltaLim : REAL; (*Upper and lower limit for the urea gian delta (-)*)
        rUreaGainDeltaRamp : REAL; (*Defines the ramp rate for urea flow adjustment (%/min)*)
        rUreaCalibFact : REAL; (*Calibration factor for the FF urea flow (-)*)
        rUreaFF_NOx_Tol : REAL; (*Defines the FF Load Table based tolerance band for the FF NOx (l/h)*)
        rTiFiltNOxFF : REAL; (*Time constant for filters used for comparison of FF LT and FF Nox (s)*)
        rUrFFNOxRampUp : REAL; (*Ramp up rate of Nox based FF in case of exceeding deviation limit to LT based FF (l/s)*)
        rUrFFNOxRampDn : REAL; (*Ramp down rate of Nox based FF in case of exceeding deviation limit to LT based FF (l/s)*)
    END_STRUCT;

   tUD_IN : STRUCT
        rT_Ch_T1LP_Avg : REAL; (*Measured ambient temperature (°C)*)
        bESCEnable : BOOL; (*Emission Supervisory Controller enabled (-)*)
        rNFlow_ESC_UreaOffs : REAL; (*Urea controller offset from Emission Supervisory Controller (ESC) controller (l/h)*)
        rCF_ESC_UreaNFlow : REAL; (*Urea controller gain correction factor send from ESC (-)*)
        rNOx_ESC_CatOut_Set : REAL; (*Reference NOx at SCR output fromm  ESC (ppm)*)
        tFlow_SCR_UreaDosingOut : tHALioAi; (*Measured urea flow (feedback signal) (l/h)*)
        tT_SCR_CatIn : tHALioAi; (*Measured exhaust gas temperature at SCR input (°C)*)
        tT_SCR_CatOut : tHALioAi; (*Measured exhaust gas temperature at SCR output (°C)*)
        rVol_Ch_Engine_Norm : REAL; (*Calculated engine volume flow (Nm3/h)*)
        rNH3_SCR_OxiIn : REAL; (*Measured ammonia (NH3) content at SCR output (ppm)*)
        tDPr_UreaDosingUnit : tHALioAi; (*Urea injection differential pressure measured (bar)*)
        rPos_SCR_UreaDosingValve : REAL; (*Urea injection valve position (%)*)
        rP_Act_Norm_Filt : REAL; (*Actual measured electric power output (% Pnom)*)
        bRel_SCR_Dosing : BOOL; (*Info from structured text to autocode that urea injection system is working and ready for operation (-)*)
        rPc_SCR_UreaDosingPump : REAL; (*Actual urea pump speed recieved from pump frequency converter in normalized speed (0..1)
Used for proper Anti-windup for urea injection control via urea pump speed control (%)*)
        tNOx_SCR_EngOut : tHALioAi; (*Measured NOx at engine output (ppm)*)
        tNOx_SCR_CatOut : tHALioAi; (*Measured NOx at SCR output (ppm)*)
        tEMLineCatOut : tUD_EMLine; (*Emissions Line (internal CEMS) Cat out (-)*)
        tEMLineOxiIn : tUD_EMLine; (*Emissions Line (internal CEMS) Oxi In (-)*)
        rNOx_SCR_CatOut_Est : REAL; (*Model based estimation of NOx at catalyst output (oxycat output) (ppm)*)
        bNOx_SCR_CatOut_Est_Ok : BOOL; (*Vailidty of model-based estimation of NOx at catalyst output (oxycat output); valid if = TRUE (-)*)
        rNOx_SCR_EngOut_Est : REAL; (*Model-based estimation of engine out NOx emissions (ppm)*)
        bNOx_SCR_EngOut_Est_Ok : BOOL; (*Validity of model-based estimation of engine out NOx emissions; valid if = True (-)*)
        rFlow_SCR_UreaDosingUnit_spMan : REAL; (*Manual command of urea flow (setpoint for UDU) (l/h)*)
        bSCR_UreaDosingUnit_Man : BOOL; (*Manual enabling/disabling of urea injection. Needs to be 1 to allow for any urea dosage controller (-)*)
        bSCR_NOxControl_Man : BOOL; (*Activate closed loop NOx control if = TRUE according to Spec Doc D2 (-)*)
        bSCR_Man : BOOL; (*G1: Manual operation mode of urea dosing system wihtout engine run Manual operation will be controlled via HMI if bSCR_Man = TRUE and autocode  dosing output will be not used in structured text. (-)*)
        bSCR_NH3SlipDetect_Blocked : BOOL; (*NH3 Slip detection blocked after 3 occurences (-)*)
        bOpModeStop : BOOL; (*Engine in stop mode (-)*)
        rHum_CatOut : REAL; (*intake air relative humiidty of humidity sensor (pu)*)
        bEMLine1_Exist : BOOL; (*SCR Emission measurement line 1 - exist (-)*)
        bEMLine2_Exist : BOOL; (*SCR Emission measurement line 2 - exist (-)*)
        rTiWaitNH3slip_fallback : REAL; (*Waiting time to switch to fallback strategy for NH3 slip detection in case of em. meas. line unavailability (s)*)
    END_STRUCT;

   tUD_OUT : STRUCT
        rFlow_SCR_UreaDosingUnit_sp : REAL; (*Urea volume flow command from urea dosage controller to urea injection system (l/h)*)
        rFlow_SCR_NOxCtrl_Y : REAL; (*Nox closed loop controller output (l/h)*)
        bSCR_NOxCtrl_Act : BOOL; (*Nox controller active (-)*)
        rNOx_SCR_NOxCtrl_act : REAL; (*Nox closed loop controller input (ppm)*)
        rNOx_SCR_CatOut_Set : REAL; (*Nox setpoint including ESC  (ppm)*)
        bSCR_EngineSteadyState : BOOL; (*Engine steady state (-)*)
        rPc_SCR_UreaDosingUnit_sp : REAL; (*Urea valve position reference (pu)*)
        rPc_SCR_UreaDosingUnit_ff : REAL; (*Urea valve position feed forwrad (pu)*)
        rPc_SCR_UreaFlowCtrl_Y : REAL; (*Urea flow closed loop controller output (-)*)
        bSCR_UreaFlowCtrl_Act : BOOL; (*Urea flow controller active (-)*)
        rFlow_SCR_UreaDosingValve_Calc : REAL; (*Inverse calculation of urea mass flow based on the actual urea dosing set-point (l/h)*)
        bSCR_NH3SlipDetected : BOOL; (*NH3 slip out of SCR catalyst detected if = TRUE (-)*)
        bSCR_NH3SlipInterrupt : BOOL; (*NH3 slip detection routine interrupted if = TRUE (-)*)
        bSCR_EMValve1_SGbOxi_Dem : BOOL; (*Switch to sampling gas position to Oxi In (-)*)
        rFlow_SCR_UreaDosingUnit_ff : REAL; (*Urea volume flow command from urea dosage controller to urea injection system feed forward (l/h)*)
        rUreaGain_Adj : REAL; (*Adjusted gain for feedforward (-)*)
        rFlow_SCR_UreaDosing_ffNH3Cor : REAL; (*Urea volume flow command from urea dosage controller feed forward corrected with the NH3 slip correction factor (l/h)*)
    END_STRUCT;

   tUD_PARA : STRUCT
        rPc_SCR_UreaSolution : REAL; (*Fraction of urea solution (%)*)
        rT_SCR_UreaDosingUnit_Release : REAL; (*U1: Lower temperature limit to start urea injection. If temperature of the catalyst is below this limit,  urea injection will be stopped. (°C)*)
        rVol_SCR_Cat : REAL; (*SCR catalyst volume (m3)*)
        rFlow_SCR_UreaDosingValveCoeff : REAL; (*Urea valve coefficient (l/h)*)
        bSCR_Active : BOOL; (*G0: The parameter is used to activate the relevant modules tasks (-)*)
        bSCR_UreaDosingValve_Exist : BOOL; (*Euqal to TRUE if dosing valve is used (-)*)
        rCF_SCR_UreaNFlowGain : REAL; (*Correction factor for feed forward load table based urea injection (-)*)
        iIdx_SCR_UreaNFlow_SelectFF : INT; (*Manual selection of preferred urea dosis calculation methid (-)*)
        bSCR_UreaFlowCtrl_Active : BOOL; (*Enables Urea injection control via speed control of urea pump (-)*)
        rNOx_SCR_CatOut_Set : REAL; (*Is taken instead of NOx sensor readings of engine out NOx measurement in case of fault sensor signals (ppm)*)
        rDNOx_SCR_NH3Slip_Hi : REAL; (*Maximum allowed NH3 slip (ppm)*)
        bSCR_NH3SlipDetect_Active : BOOL; (*Enables NH3 slip detection and control, enabled if = True (-)*)
        rNFlow_SCR_Urea30 : REAL; (*Urea dosing rate at engine load 30% (l/h)*)
        rNFlow_SCR_Urea50 : REAL; (*Urea dosing rate at engine load 50% (l/h)*)
        rNFlow_SCR_Urea75 : REAL; (*Urea dosing rate at engine load 75% (l/h)*)
        rNFlow_SCR_Urea100 : REAL; (*Urea dosing rate at engine load 100% (l/h)*)
        rA_SCR_CatSurfaceIntern : REAL; (*internal SCR catalyst surface area (m²)*)
        rSCR_NOxCtrl_Ymin : REAL; (*Minimum limitation of PID output of closed loop urea injection controller (l/h)*)
        rSCR_NOxCtrl_Ymax : REAL; (*Maximum limitation of PID output of closed loop urea injection controller (l/h)*)
        rSCR_NOxCtrl_Kd : REAL; (*Derivative gain of PID closed loop urea injection controller (-)*)
        rSCR_NOxCtrl_Ki : REAL; (*Integral gain of PID closed loop urea injection controller (l/h/ppm/s*1000)*)
        rSCR_NOxCtrl_Kp : REAL; (*proportional gain of PID closed loop urea injection controller (l/h/ppm*1000)*)
        rSCR_UreaFlowCtrl_Ymin : REAL; (*Urea valve position closed loop controller min output limit (%)*)
        rSCR_UreaFlowCtrl_Ymax : REAL; (*Urea valve position closed loop controller max output limit (%)*)
        rSCR_UreaFlowCtrl_Kd : REAL; (*Derivative gain of PIDN based urea valve closed loop controller (%/l/h*s)*)
        rSCR_UreaFlowCtrl_Ki : REAL; (*Integral gain of PIDN based urea valve closed loop controller (%/l/h/s)*)
        rSCR_UreaFlowCtrl_Kp : REAL; (*Proportional gain of PIDN based urea valve closed loop controller (%/l/h)*)
        rSCR_NOxControlWaiting : REAL; (*waiting time for NOx controller after Urea dosing activation (s)*)
        rNOx_SCR_EngOut_Expect : REAL; (*Expected Nox value  (ppm)*)
        bSCR_UreaNFlowAutoCorr_Active : BOOL; (*Automatic correction of FF enabled (-)*)
        rFlow_SCR_UreaDosingUnit_Hi : REAL; (*Dosing unit nominal flow rate (l/h)*)
        rNOx_SCR_CatOut_Hi : REAL; (*Maximum Nox CatOut (ppm)*)
        rTiSCR_EAC_DurationStartup : REAL; (*SCR Emission average calculation - duration for SCR startup (s)*)
        rTiSCR_NH3Slip_WaitNOxGrad_CL : REAL; (*Minimum wait time to restart the SCR NOx controller closed loop in case of NOx increase after NH3 slip detection (s)*)
        bFlow_SCR_UreaDosingOut_Exist : BOOL; (*SCR Urea flow rate after dosing active (-)*)
    END_STRUCT;

   tUD_PERM : STRUCT
        SM : tUD_SM_PERM; (*Perm Signal Manager ()*)
        FF : tUD_FF_PERM; (*Perm Feed Forward ()*)
        Slip : tUD_Slip_PERM; (*Perm Slip Detection ()*)
        CLNOx : tUD_CLNOx_PERM; (*Perm NOx Closed loop controller ()*)
        CLVal : tUD_CLVal_PERM; (*Perm Flow Closed loop controller (Valve) ()*)
        CLPp : tUD_CLPp_PERM; (*Perm Flow Closed loop controller (Pump) ()*)
    END_STRUCT;

   tUD_SM_DBG : STRUCT
        rNOx_SCR_CatOut_Set : REAL; (*Nox setpoint including ESC  (ppm)*)
        rNOx_EMLineCatOut : REAL; (* (ppm)*)
        bEMLineCatOut_GQ : BOOL; (* (-)*)
        rNOx_EMLineOxiIn : REAL; (* (ppm)*)
        bEMLineOxiIn_GQ : BOOL; (* (-)*)
        rNOx_SCR_NOxCtrl_act : REAL; (*Nox closed loop controller input (ppm)*)
        bFreezeCtr : BOOL; (*freeze Nox ctrl  (-)*)
        rNOx_CatOutCor : REAL; (*Nox value used for map based FF (ppm)*)
        bNOx_CatOutCor : BOOL; (* (-)*)
        rNOxEngOutCor : REAL; (* (ppm)*)
        bSCR_EngineSteadyState : BOOL; (*Steady state depending on SCR temperature and normalized electrical power (-)*)
        rTSCRAvg : REAL; (*Average SCR Cat Temperature (°C)*)
    END_STRUCT;

   tUD_SM_PERM : STRUCT
        rTiFilt_P_Act_Norm : REAL; (*Time constant of the PT1 filter for the normalized filtered power (s)*)
        rTiFilt_T_SCR_Avg : REAL; (*Time constant of the PT1 filter for the average SCR Cat temperature (s)*)
        rThresh_SS_P : REAL; (*Threshold for steady state power related (-)*)
        rThresh_SS_T_Avg : REAL; (*Threshold for steady state temperature of SCR cat (average) related (°C)*)
        rTOnDelay_SS_P : REAL; (*On-delay for the steady state power realted in terms the conditions are met (s)*)
        rTOnDelay_SS_T : REAL; (*On-delay for the steady state SCR temp. realted in terms the conditions are met (s)*)
        rP_Act_enable : REAL; (*Normalized power to enable steady state (-)*)
    END_STRUCT;

   tUD_Slip_DBG : STRUCT
        bSCR_NH3SlipDetected : BOOL; (*NH3 Slip detetcted ()*)
        rUrCorFactSlip : REAL; (*Urea flow correction factor being adjusted in case of NH3 slip detection.
Gets reduced down to zero again if no slip is detected anymore over time ()*)
        bFreezeCtrl : BOOL; (*Freeze Nox ctrl due to slip detection (-)*)
        bSCR_NH3SlipInterrupt : BOOL; (*NH3 slip detection routine interrupted (-)*)
        bNH3SlipCtrlEna : BOOL; (*Indicates if NH3 slip detection is currently enabled ()*)
        bSCR_EMValve1_SGbOxi_Dem : BOOL; (*Switch to sampling gas position to Oxi In (-)*)
    END_STRUCT;

   tUD_Slip_PERM : STRUCT
        rCemsIntFiltFact : REAL; (*First order filter time constant for NOx values averaging for slip detection and control (s)*)
        bCemsIntFiltRes : BOOL; (*Reset first order filter for NOx value filtering for NH3 slip detection and control, reset integrator if = true (-)*)
        rNH3SlipActSlope : REAL; (*Slope with which the urea correction factor for NH3 slip reduction is reduced again to zero. The higher the value, the faster the urea correction factor is eliminated again after slip detection. (1/s)*)
        rTi_SlipDetectWait : REAL; (*Waiting time before slip detection is again activated after detection completed  (s)*)
        rNOxMarginSet : REAL; (*Nox_CatOut x times higher as setpoint (-)*)
        rNOxMarginFFLT : REAL; (*Nox_CatOut x times higher as feed forward load table (-)*)
        rTiNOxMarginDelay : REAL; (*Nox higher as limit or setpoint for x seconds (s)*)
        rTiNOxCLSatDelay : REAL; (*Nox ctrl for x seconds in saturation (s)*)
        rTiSwitchValve : REAL; (*Switch over EMLine valve for x seconds (s)*)
        rGainSlipCor : REAL; (*Slip correction factor E9 (with CEMS) (-)*)
        rGainSlipCorSens : REAL; (*Slip correction factor E9a (with Nox sensor) (-)*)
        rGainFreezeCtr : REAL; (*percantege of time after slip detection, when ctrl is released again (pu)*)
        rTiWaitSteadyState : REAL; (*Wait to enable slip detection after steady state (s)*)
        rTiWaitSCRMan : REAL; (*Wait to enable slip detection after SCR manual mode (s)*)
        rTiWaitSwitch : REAL; (*Wait to enable slip detection after switch valve over to OxiIn (s)*)
        rTiFilter_Nox : REAL; (*Filter constant for Nox derivative (s)*)
        rNOxGradLim : REAL; (*Nox gradient limit to unfreeze controller (ppm/s)*)
        rNOxFactorSet_CL : REAL; (*Nox_CatOut x times lower than setpoint to restart closed loop controller during NH3 slip correction routine (-)*)
    END_STRUCT;
END_TYPE
TYPE
rtB_Cell1_UDC : STRUCT
	DiscreteTimeIntegrator : REAL;
	LookupTableDynamic : REAL;
END_STRUCT;
rtDW_Cell1_UDC : STRUCT
	DiscreteTimeIntegrator_DSTATE : REAL;
	DiscreteTimeIntegrator_PrevRese : SINT;
	DiscreteTimeIntegrator_IC_LOADI : USINT;
END_STRUCT;
rtB_Filter_UDC : STRUCT
	Switch : REAL;
END_STRUCT;
rtDW_Filter_UDC : STRUCT
	DiscreteTimeIntegrator_DSTATE : REAL;
	DiscreteTimeIntegrator_PrevRese : SINT;
	DiscreteTimeIntegrator_IC_LOADI : USINT;
END_STRUCT;
rtB_TON_UDC : STRUCT
	LogicalOperator3 : BOOL;
END_STRUCT;
rtDW_TON_UDC : STRUCT
	DiscreteTimeIntegrator_DSTATE : REAL;
	DiscreteTimeIntegrator_PrevRese : SINT;
END_STRUCT;
rtB_TP_UDC : STRUCT
	Merge : REAL;
	LogicalOperator1 : BOOL;
END_STRUCT;
rtDW_TP_UDC : STRUCT
	DelayInput2_DSTATE : REAL;
	UnitDelay2_DSTATE : BOOL;
END_STRUCT;
rtB_TOF_UDC : STRUCT
	LogicalOperator1 : BOOL;
END_STRUCT;
rtDW_TOF_UDC : STRUCT
	DiscreteTimeIntegrator_DSTATE : LREAL;
	DiscreteTimeIntegrator_PrevRese : SINT;
	DiscreteTimeIntegrator_IC_LOADI : USINT;
END_STRUCT;
BlockIO_UDC : STRUCT
	BusInput2 : tUD_PERM;
	BusInput : tUD_IN;
	BusInput1 : tUD_PARA;
	Merge5 : ARRAY[0..3] OF REAL;
	UnitDelay : UDINT;
	TON_p : rtB_TON_UDC;
	TON3_p : rtB_TON_UDC;
	TON2_a : rtB_TON_UDC;
	TON1_p : rtB_TON_UDC;
	TON_fg : rtB_TON_UDC;
	TP_m : rtB_TP_UDC;
	TON_o : rtB_TON_UDC;
	Filter_OxiIn : rtB_Filter_UDC;
	Filter_CatOut : rtB_Filter_UDC;
	TP1 : rtB_TP_UDC;
	TON2 : rtB_TON_UDC;
	TON1_k : rtB_TON_UDC;
	TON_i : rtB_TON_UDC;
	TP_e : rtB_TP_UDC;
	TON3 : rtB_TON_UDC;
	TON_a : rtB_TON_UDC;
	TON1 : rtB_TON_UDC;
	TON : rtB_TON_UDC;
	Filter2 : rtB_Filter_UDC;
	Filter : rtB_Filter_UDC;
	TOF1 : rtB_TOF_UDC;
	TOF : rtB_TOF_UDC;
	TON_f : rtB_TON_UDC;
	Filter_DPr_h : rtB_Filter_UDC;
	Filter_DPr : rtB_Filter_UDC;
	TP : rtB_TP_UDC;
	TON_j : rtB_TON_UDC;
	Filter1 : rtB_Filter_UDC;
	Filter_o : rtB_Filter_UDC;
	Cell3 : rtB_Cell1_UDC;
	Cell2 : rtB_Cell1_UDC;
	Cell1 : rtB_Cell1_UDC;
END_STRUCT;
D_Work_UDC : STRUCT
	Delay_DSTATE : REAL;
	Delay_DSTATE_d : REAL;
	DiscreteTimeIntegrator_DSTATE : REAL;
	DiscreteTimeIntegrator_DSTATE_i : REAL;
	VariableIntegerDelay_DSTATE : ARRAY[0..999] OF REAL;
	UnitDelay_DSTATE : REAL;
	DiscreteTimeIntegrator_DSTATE_p : REAL;
	DiscreteTimeIntegrator1_DSTATE : REAL;
	UnitDelay_DSTATE_g : REAL;
	UnitDelay4_DSTATE : REAL;
	Delay_DSTATE_k : REAL;
	Delay_DSTATE_h : REAL;
	DiscreteTimeIntegrator_DSTATE_o : REAL;
	Delay_DSTATE_f : REAL;
	DiscreteTimeIntegrator_DSTATE_d : REAL;
	DiscreteTimeIntegrator1_DSTAT_l : REAL;
	UnitDelay_DSTATE_j : REAL;
	DiscreteTimeIntegrator_DSTATE_e : REAL;
	DiscreteTimeIntegrator1_DSTAT_b : REAL;
	UnitDelay_DSTATE_n : REAL;
	UnitDelay_DSTATE_d : REAL;
	UnitDelay2_DSTATE : REAL;
	UnitDelay_DSTATE_c : UDINT;
	rNOx_EMLineCatOut_1 : REAL;
	rNOx_EMLineOxiIn_1 : REAL;
	rNOx_Act_1 : REAL;
	UnitDelay4_DSTATE_j : BOOL;
	UnitDelay_DSTATE_l : BOOL;
	DelayInput1_DSTATE : BOOL;
	UnitDelay_DSTATE_dg : BOOL;
	UnitDelay2_DSTATE_f : BOOL;
	UnitDelay2_DSTATE_i : BOOL;
	DelayInput1_DSTATE_m : BOOL;
	UnitDelay_DSTATE_jw : BOOL;
	DiscreteTimeIntegrator_PrevRese : SINT;
	DiscreteTimeIntegrator_PrevRe_k : SINT;
	DiscreteTimeIntegrator_PrevRe_j : SINT;
	DiscreteTimeIntegrator1_PrevRes : SINT;
	DiscreteTimeIntegrator_PrevRe_e : SINT;
	DiscreteTimeIntegrator_PrevR_j5 : SINT;
	DiscreteTimeIntegrator1_PrevR_b : SINT;
	DiscreteTimeIntegrator_PrevRe_p : SINT;
	DiscreteTimeIntegrator1_PrevR_e : SINT;
	icLoad : USINT;
	DiscreteTimeIntegrator_IC_LOADI : USINT;
	DiscreteTimeIntegrator1_IC_LOAD : USINT;
	icLoad_g : USINT;
	icLoad_e : USINT;
	icLoad_d : USINT;
	DiscreteTimeIntegrator_IC_LOA_e : USINT;
	DiscreteTimeIntegrator1_IC_LO_n : USINT;
	DiscreteTimeIntegrator_IC_LOA_f : USINT;
	DiscreteTimeIntegrator1_IC_LO_i : USINT;
	Memory_PreviousInput : BOOL;
	Relay1_Mode : BOOL;
	Memory_PreviousInput_k : BOOL;
	x : BOOL;
	rNOx_EMLineCatOut_1_not_empty : BOOL;
	rNOx_EMLineOxiIn_1_not_empty : BOOL;
	rNOx_Act_1_not_empty : BOOL;
	TON_p : rtDW_TON_UDC;
	TON3_p : rtDW_TON_UDC;
	TON2_a : rtDW_TON_UDC;
	TON1_p : rtDW_TON_UDC;
	TON_fg : rtDW_TON_UDC;
	TP_m : rtDW_TP_UDC;
	TON_o : rtDW_TON_UDC;
	Filter_OxiIn : rtDW_Filter_UDC;
	Filter_CatOut : rtDW_Filter_UDC;
	TP1 : rtDW_TP_UDC;
	TON2 : rtDW_TON_UDC;
	TON1_k : rtDW_TON_UDC;
	TON_i : rtDW_TON_UDC;
	TP_e : rtDW_TP_UDC;
	TON3 : rtDW_TON_UDC;
	TON_a : rtDW_TON_UDC;
	TON1 : rtDW_TON_UDC;
	TON : rtDW_TON_UDC;
	Filter2 : rtDW_Filter_UDC;
	Filter : rtDW_Filter_UDC;
	TOF1 : rtDW_TOF_UDC;
	TOF : rtDW_TOF_UDC;
	TON_f : rtDW_TON_UDC;
	Filter_DPr_h : rtDW_Filter_UDC;
	Filter_DPr : rtDW_Filter_UDC;
	TP : rtDW_TP_UDC;
	TON_j : rtDW_TON_UDC;
	Filter1 : rtDW_Filter_UDC;
	Filter_o : rtDW_Filter_UDC;
	Cell3 : rtDW_Cell1_UDC;
	Cell2 : rtDW_Cell1_UDC;
	Cell1 : rtDW_Cell1_UDC;
END_STRUCT;
PrevZCSigStates_UDC : STRUCT
	Delay_Reset_ZCE : USINT;
	Delay_Reset_ZCE_n : USINT;
	Delay_Reset_ZCE_d : USINT;
	Delay_Reset_ZCE_i : USINT;
	Delay_Reset_ZCE_b : USINT;
END_STRUCT;
rtC_Filter_UDC : STRUCT
	Conversion : REAL;
END_STRUCT;
ConstBlockIO_UDC : STRUCT
	Filter_OxiIn : rtC_Filter_UDC;
	Filter_CatOut : rtC_Filter_UDC;
	Filter2 : rtC_Filter_UDC;
	Filter : rtC_Filter_UDC;
	Filter_DPr_h : rtC_Filter_UDC;
	Filter_DPr : rtC_Filter_UDC;
	Filter1 : rtC_Filter_UDC;
	Filter_o : rtC_Filter_UDC;
END_STRUCT;
ConstParam_UDC : STRUCT
	Constant_Value : ARRAY[0..4] OF LREAL;
	InterpolationUsingPre : ARRAY[0..1] OF UDINT;
	pooled28 : ARRAY[0..15] OF BOOL;
END_STRUCT;
ExternalInputs_UDC : STRUCT
	InUD : tUD_IN;
	ParaUD : tUD_PARA;
	PermUD : tUD_PERM;
END_STRUCT;
ExternalOutputs_UDC : STRUCT
	OutUDbus : tUD_OUT;
	DebugUDbus : tUD_DBG;
END_STRUCT;
tag_RTM_UDC : STRUCT
	errorStatus : REFERENCE TO USINT;
END_STRUCT;
END_TYPE
```

#### UDC.h
```c
/********************************************************************
 * COPYRIGHT -- Bernecker + Rainer Industrie-Elektronik Ges.m.b.H.
 ********************************************************************
 * Program: UDC
 * File: UDC.h
 * Author: 105055527
 * Created: Thu Mar 02 16:51:06 2017
 ********************************************************************
 * Header for program UDC
 ********************************************************************
 * Generated with B&R Automation Studio Target for Simulink V4.2
 * (ERT based)
 ********************************************************************/

#ifndef RTW_HEADER_UDC_h_
#define RTW_HEADER_UDC_h_
#ifndef UDC_COMMON_INCLUDES_
# define UDC_COMMON_INCLUDES_
#include <math.h>
#include "rtwtypes.h"
#include "rtGetInf.h"
#include "rtGetNaN.h"
#include "rt_nonfinite.h"
#endif                                 /* UDC_COMMON_INCLUDES_ */

#include "UDC_types.h"
#include "lUDC.h"

/* Macros for accessing real-time model data structure */
#ifndef rtmGetErrorStatus
# define rtmGetErrorStatus(rtm)        ((rtm)->errorStatus)
#endif

#ifndef rtmSetErrorStatus
# define rtmSetErrorStatus(rtm, val)   ((rtm)->errorStatus = (val))
#endif

#ifndef rtmGetStopRequested
# define rtmGetStopRequested(rtm)      ((void*) 0)
#endif

#ifndef MIN
#define MIN(a,b)                       ((a) < (b) ? (a) : (b))
#endif

#ifndef MAX
#define MAX(a,b)                       ((a) > (b) ? (a) : (b))
#endif

/* Block signals for system '<S30>/Cell1' */

/* Block states (auto storage) for system '<S30>/Cell1' */

/* Block signals for system '<S15>/Filter' */

/* Block states (auto storage) for system '<S15>/Filter' */

/* Block signals for system '<S65>/TON' */

/* Block states (auto storage) for system '<S65>/TON' */

/* Block signals for system '<S65>/TP' */

/* Block states (auto storage) for system '<S65>/TP' */

/* Block signals for system '<S119>/TOF' */

/* Block states (auto storage) for system '<S119>/TOF' */

/* Block signals (auto storage) */

/* Block states (auto storage) for system '<Root>' */

/* Zero-crossing (trigger) state */

/* Invariant block signals for system '<S15>/Filter' */

/* Invariant block signals (auto storage) */

/* Constant parameters (auto storage) */

/* External inputs (root inport signals with auto storage) */

/* External outputs (root outports fed by signals with auto storage) */

/* Real-time Model Data Structure */

/* Block signals (auto storage) */
extern BlockIO_UDC UDC_B;

/* Block states (auto storage) */
extern D_Work_UDC UDC_DWork;

/* External inputs (root inport signals with auto storage) */
extern ExternalInputs_UDC UDC_U;

/* External outputs (root outports fed by signals with auto storage) */
extern ExternalOutputs_UDC UDC_Y;
extern const ConstBlockIO_UDC UDC_ConstB;/* constant block i/o */

/* Constant parameters (auto storage) */
extern const ConstParam_UDC UDC_ConstP;

/* Model entry point functions */
extern void UDC_initialize(struct fUDC* inst);
extern void UDC_step(struct fUDC* inst);
extern void UDC_terminate(struct fUDC* inst);

/* Real-time Model object */
extern RT_MODEL_UDC *const UDC_M;

/*-
 * The generated code includes comments that allow you to trace directly
 * back to the appropriate location in the model.  The basic format
 * is <system>/block_name, where system is the system number (uniquely
 * assigned by Simulink) and block_name is the name of the block.
 *
 * Use the MATLAB hilite_system command to trace the generated code back
 * to the model.  For example,
 *
 * hilite_system('<S3>')    - opens system 3
 * hilite_system('<S3>/Kp') - opens and selects block Kp which resides in S3
 *
 * Here is the system hierarchy for this model
 *
 * '<Root>' : 'UDC'
 * '<S1>'   : 'UDC/DocBlock1'
 * '<S2>'   : 'UDC/Environment Controller'
 * '<S3>'   : 'UDC/Environment Controller1'
 * '<S4>'   : 'UDC/Environment Controller2'
 * '<S5>'   : 'UDC/FeedForward'
 * '<S6>'   : 'UDC/Flow_CL'
 * '<S7>'   : 'UDC/Info1'
 * '<S8>'   : 'UDC/NOx_CL'
 * '<S9>'   : 'UDC/SignalManager'
 * '<S10>'  : 'UDC/SlipDetection'
 * '<S11>'  : 'UDC/FeedForward/D1_FF_Manager'
 * '<S12>'  : 'UDC/FeedForward/D1a_FF_LoadTab'
 * '<S13>'  : 'UDC/FeedForward/D1b_FF_NOx'
 * '<S14>'  : 'UDC/FeedForward/D1c_FF_map'
 * '<S15>'  : 'UDC/FeedForward/D6_FF_Adjust'
 * '<S16>'  : 'UDC/FeedForward/FF_NH3Sens_based'
 * '<S17>'  : 'UDC/FeedForward/spaceVelocityCalc'
 * '<S18>'  : 'UDC/FeedForward/D1_FF_Manager/ESC_Corr'
 * '<S19>'  : 'UDC/FeedForward/D1_FF_Manager/Saturation Dynamic1'
 * '<S20>'  : 'UDC/FeedForward/D1_FF_Manager/UrInFFCalcManager'
 * '<S21>'  : 'UDC/FeedForward/D1_FF_Manager/UrInFFCalcManager/UrInMethCalculation'
 * '<S22>'  : 'UDC/FeedForward/D1b_FF_NOx/Divisor'
 * '<S23>'  : 'UDC/FeedForward/D1b_FF_NOx/Divisor1'
 * '<S24>'  : 'UDC/FeedForward/D1b_FF_NOx/Divisor2'
 * '<S25>'  : 'UDC/FeedForward/D1b_FF_NOx/Divisor/Data Type Conversion Inherited'
 * '<S26>'  : 'UDC/FeedForward/D1b_FF_NOx/Divisor1/Data Type Conversion Inherited'
 * '<S27>'  : 'UDC/FeedForward/D1b_FF_NOx/Divisor2/Data Type Conversion Inherited'
 * '<S28>'  : 'UDC/FeedForward/D1c_FF_map/SCRStorageDynamics'
 * '<S29>'  : 'UDC/FeedForward/D1c_FF_map/SCRStorageDynamicsNOxInclude'
 * '<S30>'  : 'UDC/FeedForward/D1c_FF_map/SCRThermalMaxStorageModel'
 * '<S31>'  : 'UDC/FeedForward/D1c_FF_map/Saturation Dynamic1'
 * '<S32>'  : 'UDC/FeedForward/D1c_FF_map/Saturation Dynamic2'
 * '<S33>'  : 'UDC/FeedForward/D1c_FF_map/Saturation Dynamic3'
 * '<S34>'  : 'UDC/FeedForward/D1c_FF_map/UreaMassFlowCalcFF'
 * '<S35>'  : 'UDC/FeedForward/D1c_FF_map/steadyStateUsageMap'
 * '<S36>'  : 'UDC/FeedForward/D1c_FF_map/SCRThermalMaxStorageModel/Cell1'
 * '<S37>'  : 'UDC/FeedForward/D1c_FF_map/SCRThermalMaxStorageModel/Cell2'
 * '<S38>'  : 'UDC/FeedForward/D1c_FF_map/SCRThermalMaxStorageModel/Cell3'
 * '<S39>'  : 'UDC/FeedForward/D1c_FF_map/SCRThermalMaxStorageModel/Divisor'
 * '<S40>'  : 'UDC/FeedForward/D1c_FF_map/SCRThermalMaxStorageModel/Cell1/Divisor'
 * '<S41>'  : 'UDC/FeedForward/D1c_FF_map/SCRThermalMaxStorageModel/Cell1/Divisor1'
 * '<S42>'  : 'UDC/FeedForward/D1c_FF_map/SCRThermalMaxStorageModel/Cell1/Divisor/Data Type Conversion Inherited'
 * '<S43>'  : 'UDC/FeedForward/D1c_FF_map/SCRThermalMaxStorageModel/Cell1/Divisor1/Data Type Conversion Inherited'
 * '<S44>'  : 'UDC/FeedForward/D1c_FF_map/SCRThermalMaxStorageModel/Cell2/Divisor'
 * '<S45>'  : 'UDC/FeedForward/D1c_FF_map/SCRThermalMaxStorageModel/Cell2/Divisor1'
 * '<S46>'  : 'UDC/FeedForward/D1c_FF_map/SCRThermalMaxStorageModel/Cell2/Divisor/Data Type Conversion Inherited'
 * '<S47>'  : 'UDC/FeedForward/D1c_FF_map/SCRThermalMaxStorageModel/Cell2/Divisor1/Data Type Conversion Inherited'
 * '<S48>'  : 'UDC/FeedForward/D1c_FF_map/SCRThermalMaxStorageModel/Cell3/Divisor'
 * '<S49>'  : 'UDC/FeedForward/D1c_FF_map/SCRThermalMaxStorageModel/Cell3/Divisor1'
 * '<S50>'  : 'UDC/FeedForward/D1c_FF_map/SCRThermalMaxStorageModel/Cell3/Divisor/Data Type Conversion Inherited'
 * '<S51>'  : 'UDC/FeedForward/D1c_FF_map/SCRThermalMaxStorageModel/Cell3/Divisor1/Data Type Conversion Inherited'
 * '<S52>'  : 'UDC/FeedForward/D1c_FF_map/SCRThermalMaxStorageModel/Divisor/Data Type Conversion Inherited'
 * '<S53>'  : 'UDC/FeedForward/D1c_FF_map/UreaMassFlowCalcFF/Divisor'
 * '<S54>'  : 'UDC/FeedForward/D1c_FF_map/UreaMassFlowCalcFF/Divisor1'
 * '<S55>'  : 'UDC/FeedForward/D1c_FF_map/UreaMassFlowCalcFF/Divisor2'
 * '<S56>'  : 'UDC/FeedForward/D1c_FF_map/UreaMassFlowCalcFF/Divisor/Data Type Conversion Inherited'
 * '<S57>'  : 'UDC/FeedForward/D1c_FF_map/UreaMassFlowCalcFF/Divisor1/Data Type Conversion Inherited'
 * '<S58>'  : 'UDC/FeedForward/D1c_FF_map/UreaMassFlowCalcFF/Divisor2/Data Type Conversion Inherited'
 * '<S59>'  : 'UDC/FeedForward/D1c_FF_map/steadyStateUsageMap/SV_TSCR_to_NOxRedRatio'
 * '<S60>'  : 'UDC/FeedForward/D1c_FF_map/steadyStateUsageMap/Saturation Dynamic'
 * '<S61>'  : 'UDC/FeedForward/D6_FF_Adjust/Divisor1'
 * '<S62>'  : 'UDC/FeedForward/D6_FF_Adjust/Filter'
 * '<S63>'  : 'UDC/FeedForward/D6_FF_Adjust/Filter1'
 * '<S64>'  : 'UDC/FeedForward/D6_FF_Adjust/Saturation Dynamic1'
 * '<S65>'  : 'UDC/FeedForward/D6_FF_Adjust/Timing'
 * '<S66>'  : 'UDC/FeedForward/D6_FF_Adjust/rateLimit'
 * '<S67>'  : 'UDC/FeedForward/D6_FF_Adjust/Divisor1/Data Type Conversion Inherited'
 * '<S68>'  : 'UDC/FeedForward/D6_FF_Adjust/Filter/Divisor'
 * '<S69>'  : 'UDC/FeedForward/D6_FF_Adjust/Filter/Divisor/Data Type Conversion Inherited'
 * '<S70>'  : 'UDC/FeedForward/D6_FF_Adjust/Filter1/Divisor'
 * '<S71>'  : 'UDC/FeedForward/D6_FF_Adjust/Filter1/Divisor/Data Type Conversion Inherited'
 * '<S72>'  : 'UDC/FeedForward/D6_FF_Adjust/Timing/TON'
 * '<S73>'  : 'UDC/FeedForward/D6_FF_Adjust/Timing/TP'
 * '<S74>'  : 'UDC/FeedForward/D6_FF_Adjust/Timing/TON/Data Type Conversion Inherited'
 * '<S75>'  : 'UDC/FeedForward/D6_FF_Adjust/Timing/TP/Compare To Zero'
 * '<S76>'  : 'UDC/FeedForward/D6_FF_Adjust/Timing/TP/Enabled Subsystem'
 * '<S77>'  : 'UDC/FeedForward/D6_FF_Adjust/Timing/TP/Enabled Subsystem1'
 * '<S78>'  : 'UDC/FeedForward/D6_FF_Adjust/Timing/TP/Rate Limiter'
 * '<S79>'  : 'UDC/FeedForward/D6_FF_Adjust/Timing/TP/Rate Limiter/Saturation Dynamic'
 * '<S80>'  : 'UDC/FeedForward/D6_FF_Adjust/rateLimit/Saturation Dynamic'
 * '<S81>'  : 'UDC/FeedForward/FF_NH3Sens_based/Saturation Dynamic'
 * '<S82>'  : 'UDC/FeedForward/spaceVelocityCalc/Divisor1'
 * '<S83>'  : 'UDC/FeedForward/spaceVelocityCalc/Divisor1/Data Type Conversion Inherited'
 * '<S84>'  : 'UDC/Flow_CL/Dummy'
 * '<S85>'  : 'UDC/Flow_CL/UrPumpCntr'
 * '<S86>'  : 'UDC/Flow_CL/UrValCntr'
 * '<S87>'  : 'UDC/Flow_CL/UrPumpCntr/Divisor1'
 * '<S88>'  : 'UDC/Flow_CL/UrPumpCntr/PID_UrPump'
 * '<S89>'  : 'UDC/Flow_CL/UrPumpCntr/PumpFlowCorrCheck'
 * '<S90>'  : 'UDC/Flow_CL/UrPumpCntr/Saturation Dynamic1'
 * '<S91>'  : 'UDC/Flow_CL/UrPumpCntr/Saturation Dynamic2'
 * '<S92>'  : 'UDC/Flow_CL/UrPumpCntr/Divisor1/Data Type Conversion Inherited'
 * '<S93>'  : 'UDC/Flow_CL/UrValCntr/Divisor1'
 * '<S94>'  : 'UDC/Flow_CL/UrValCntr/PID_UrVal'
 * '<S95>'  : 'UDC/Flow_CL/UrValCntr/Saturation Dynamic1'
 * '<S96>'  : 'UDC/Flow_CL/UrValCntr/Saturation Dynamic2'
 * '<S97>'  : 'UDC/Flow_CL/UrValCntr/U6_ValveFlowCorr'
 * '<S98>'  : 'UDC/Flow_CL/UrValCntr/ValveFlowCorrCheck'
 * '<S99>'  : 'UDC/Flow_CL/UrValCntr/Divisor1/Data Type Conversion Inherited'
 * '<S100>' : 'UDC/Flow_CL/UrValCntr/U6_ValveFlowCorr/Divisor'
 * '<S101>' : 'UDC/Flow_CL/UrValCntr/U6_ValveFlowCorr/Filter_DPr'
 * '<S102>' : 'UDC/Flow_CL/UrValCntr/U6_ValveFlowCorr/Divisor/Data Type Conversion Inherited'
 * '<S103>' : 'UDC/Flow_CL/UrValCntr/U6_ValveFlowCorr/Filter_DPr/Divisor'
 * '<S104>' : 'UDC/Flow_CL/UrValCntr/U6_ValveFlowCorr/Filter_DPr/Divisor/Data Type Conversion Inherited'
 * '<S105>' : 'UDC/Flow_CL/UrValCntr/ValveFlowCorrCheck/Divisor2'
 * '<S106>' : 'UDC/Flow_CL/UrValCntr/ValveFlowCorrCheck/Filter_DPr'
 * '<S107>' : 'UDC/Flow_CL/UrValCntr/ValveFlowCorrCheck/Divisor2/Data Type Conversion Inherited'
 * '<S108>' : 'UDC/Flow_CL/UrValCntr/ValveFlowCorrCheck/Filter_DPr/Divisor'
 * '<S109>' : 'UDC/Flow_CL/UrValCntr/ValveFlowCorrCheck/Filter_DPr/Divisor/Data Type Conversion Inherited'
 * '<S110>' : 'UDC/NOx_CL/Saturation Dynamic1'
 * '<S111>' : 'UDC/NOx_CL/UreaInjectionClosedLoopControl'
 * '<S112>' : 'UDC/NOx_CL/UreaInjectionClosedLoopControl/PID_NOx'
 * '<S113>' : 'UDC/NOx_CL/UreaInjectionClosedLoopControl/PID_Para'
 * '<S114>' : 'UDC/NOx_CL/UreaInjectionClosedLoopControl/Saturation Dynamic1'
 * '<S115>' : 'UDC/NOx_CL/UreaInjectionClosedLoopControl/Saturation Dynamic2'
 * '<S116>' : 'UDC/NOx_CL/UreaInjectionClosedLoopControl/TON'
 * '<S117>' : 'UDC/NOx_CL/UreaInjectionClosedLoopControl/TON/Data Type Conversion Inherited'
 * '<S118>' : 'UDC/SignalManager/E20_NOxEngOutManager'
 * '<S119>' : 'UDC/SignalManager/E21_NOxCatOutManager'
 * '<S120>' : 'UDC/SignalManager/E22_Engine_Cat_SteadyState'
 * '<S121>' : 'UDC/SignalManager/E23_T_SCR_Avg'
 * '<S122>' : 'UDC/SignalManager/E21_NOxCatOutManager/MATLAB Function'
 * '<S123>' : 'UDC/SignalManager/E21_NOxCatOutManager/TOF'
 * '<S124>' : 'UDC/SignalManager/E21_NOxCatOutManager/TOF1'
 * '<S125>' : 'UDC/SignalManager/E21_NOxCatOutManager/TOF/Data Type Conversion Inherited'
 * '<S126>' : 'UDC/SignalManager/E21_NOxCatOutManager/TOF1/Data Type Conversion Inherited'
 * '<S127>' : 'UDC/SignalManager/E22_Engine_Cat_SteadyState/Filter'
 * '<S128>' : 'UDC/SignalManager/E22_Engine_Cat_SteadyState/Filter2'
 * '<S129>' : 'UDC/SignalManager/E22_Engine_Cat_SteadyState/TON'
 * '<S130>' : 'UDC/SignalManager/E22_Engine_Cat_SteadyState/TON1'
 * '<S131>' : 'UDC/SignalManager/E22_Engine_Cat_SteadyState/Filter/Divisor'
 * '<S132>' : 'UDC/SignalManager/E22_Engine_Cat_SteadyState/Filter/Divisor/Data Type Conversion Inherited'
 * '<S133>' : 'UDC/SignalManager/E22_Engine_Cat_SteadyState/Filter2/Divisor'
 * '<S134>' : 'UDC/SignalManager/E22_Engine_Cat_SteadyState/Filter2/Divisor/Data Type Conversion Inherited'
 * '<S135>' : 'UDC/SignalManager/E22_Engine_Cat_SteadyState/TON/Data Type Conversion Inherited'
 * '<S136>' : 'UDC/SignalManager/E22_Engine_Cat_SteadyState/TON1/Data Type Conversion Inherited'
 * '<S137>' : 'UDC/SlipDetection/E9_1_SlipCtrlEna'
 * '<S138>' : 'UDC/SlipDetection/E9_2'
 * '<S139>' : 'UDC/SlipDetection/E9_3_SlipDetection'
 * '<S140>' : 'UDC/SlipDetection/E9_4_SlipDetection'
 * '<S141>' : 'UDC/SlipDetection/E9_5_SlipCtrlCorr'
 * '<S142>' : 'UDC/SlipDetection/E9_1_SlipCtrlEna/Detect Decrease'
 * '<S143>' : 'UDC/SlipDetection/E9_1_SlipCtrlEna/TOF'
 * '<S144>' : 'UDC/SlipDetection/E9_1_SlipCtrlEna/TON'
 * '<S145>' : 'UDC/SlipDetection/E9_1_SlipCtrlEna/TON3'
 * '<S146>' : 'UDC/SlipDetection/E9_1_SlipCtrlEna/TP'
 * '<S147>' : 'UDC/SlipDetection/E9_1_SlipCtrlEna/TOF/rateLimit'
 * '<S148>' : 'UDC/SlipDetection/E9_1_SlipCtrlEna/TOF/rateLimit/Saturation Dynamic'
 * '<S149>' : 'UDC/SlipDetection/E9_1_SlipCtrlEna/TON/Data Type Conversion Inherited'
 * '<S150>' : 'UDC/SlipDetection/E9_1_SlipCtrlEna/TON3/Data Type Conversion Inherited'
 * '<S151>' : 'UDC/SlipDetection/E9_1_SlipCtrlEna/TP/Compare To Zero'
 * '<S152>' : 'UDC/SlipDetection/E9_1_SlipCtrlEna/TP/Enabled Subsystem'
 * '<S153>' : 'UDC/SlipDetection/E9_1_SlipCtrlEna/TP/Enabled Subsystem1'
 * '<S154>' : 'UDC/SlipDetection/E9_1_SlipCtrlEna/TP/Rate Limiter'
 * '<S155>' : 'UDC/SlipDetection/E9_1_SlipCtrlEna/TP/Rate Limiter/Saturation Dynamic'
 * '<S156>' : 'UDC/SlipDetection/E9_2/S-R Flip-Flop'
 * '<S157>' : 'UDC/SlipDetection/E9_2/TON'
 * '<S158>' : 'UDC/SlipDetection/E9_2/TON1'
 * '<S159>' : 'UDC/SlipDetection/E9_2/TON2'
 * '<S160>' : 'UDC/SlipDetection/E9_2/TP1'
 * '<S161>' : 'UDC/SlipDetection/E9_2/TON/Data Type Conversion Inherited'
 * '<S162>' : 'UDC/SlipDetection/E9_2/TON1/Data Type Conversion Inherited'
 * '<S163>' : 'UDC/SlipDetection/E9_2/TON2/Data Type Conversion Inherited'
 * '<S164>' : 'UDC/SlipDetection/E9_2/TP1/Compare To Zero'
 * '<S165>' : 'UDC/SlipDetection/E9_2/TP1/Enabled Subsystem'
 * '<S166>' : 'UDC/SlipDetection/E9_2/TP1/Enabled Subsystem1'
 * '<S167>' : 'UDC/SlipDetection/E9_2/TP1/Rate Limiter'
 * '<S168>' : 'UDC/SlipDetection/E9_2/TP1/Rate Limiter/Saturation Dynamic'
 * '<S169>' : 'UDC/SlipDetection/E9_3_SlipDetection/Compare To Zero'
 * '<S170>' : 'UDC/SlipDetection/E9_3_SlipDetection/Divisor'
 * '<S171>' : 'UDC/SlipDetection/E9_3_SlipDetection/Filter_CatOut'
 * '<S172>' : 'UDC/SlipDetection/E9_3_SlipDetection/Filter_OxiIn'
 * '<S173>' : 'UDC/SlipDetection/E9_3_SlipDetection/TON'
 * '<S174>' : 'UDC/SlipDetection/E9_3_SlipDetection/TP'
 * '<S175>' : 'UDC/SlipDetection/E9_3_SlipDetection/Divisor/Data Type Conversion Inherited'
 * '<S176>' : 'UDC/SlipDetection/E9_3_SlipDetection/Filter_CatOut/Divisor'
 * '<S177>' : 'UDC/SlipDetection/E9_3_SlipDetection/Filter_CatOut/Divisor/Data Type Conversion Inherited'
 * '<S178>' : 'UDC/SlipDetection/E9_3_SlipDetection/Filter_OxiIn/Divisor'
 * '<S179>' : 'UDC/SlipDetection/E9_3_SlipDetection/Filter_OxiIn/Divisor/Data Type Conversion Inherited'
 * '<S180>' : 'UDC/SlipDetection/E9_3_SlipDetection/TON/Data Type Conversion Inherited'
 * '<S181>' : 'UDC/SlipDetection/E9_3_SlipDetection/TP/Compare To Zero'
 * '<S182>' : 'UDC/SlipDetection/E9_3_SlipDetection/TP/Enabled Subsystem'
 * '<S183>' : 'UDC/SlipDetection/E9_3_SlipDetection/TP/Enabled Subsystem1'
 * '<S184>' : 'UDC/SlipDetection/E9_3_SlipDetection/TP/Rate Limiter'
 * '<S185>' : 'UDC/SlipDetection/E9_3_SlipDetection/TP/Rate Limiter/Saturation Dynamic'
 * '<S186>' : 'UDC/SlipDetection/E9_4_SlipDetection/Divisor2'
 * '<S187>' : 'UDC/SlipDetection/E9_4_SlipDetection/TON'
 * '<S188>' : 'UDC/SlipDetection/E9_4_SlipDetection/TON1'
 * '<S189>' : 'UDC/SlipDetection/E9_4_SlipDetection/TON2'
 * '<S190>' : 'UDC/SlipDetection/E9_4_SlipDetection/TON3'
 * '<S191>' : 'UDC/SlipDetection/E9_4_SlipDetection/Divisor2/Data Type Conversion Inherited'
 * '<S192>' : 'UDC/SlipDetection/E9_4_SlipDetection/TON/Data Type Conversion Inherited'
 * '<S193>' : 'UDC/SlipDetection/E9_4_SlipDetection/TON1/Data Type Conversion Inherited'
 * '<S194>' : 'UDC/SlipDetection/E9_4_SlipDetection/TON2/Data Type Conversion Inherited'
 * '<S195>' : 'UDC/SlipDetection/E9_4_SlipDetection/TON3/Data Type Conversion Inherited'
 * '<S196>' : 'UDC/SlipDetection/E9_5_SlipCtrlCorr/Compare To Constant'
 * '<S197>' : 'UDC/SlipDetection/E9_5_SlipCtrlCorr/Compare To Constant1'
 * '<S198>' : 'UDC/SlipDetection/E9_5_SlipCtrlCorr/Detect Rise Positive'
 * '<S199>' : 'UDC/SlipDetection/E9_5_SlipCtrlCorr/Filter1'
 * '<S200>' : 'UDC/SlipDetection/E9_5_SlipCtrlCorr/S-R Flip-Flop'
 * '<S201>' : 'UDC/SlipDetection/E9_5_SlipCtrlCorr/TON'
 * '<S202>' : 'UDC/SlipDetection/E9_5_SlipCtrlCorr/rateLimit'
 * '<S203>' : 'UDC/SlipDetection/E9_5_SlipCtrlCorr/rateLimit1'
 * '<S204>' : 'UDC/SlipDetection/E9_5_SlipCtrlCorr/switchHold fct1'
 * '<S205>' : 'UDC/SlipDetection/E9_5_SlipCtrlCorr/Detect Rise Positive/Positive'
 * '<S206>' : 'UDC/SlipDetection/E9_5_SlipCtrlCorr/Filter1/Divisor'
 * '<S207>' : 'UDC/SlipDetection/E9_5_SlipCtrlCorr/Filter1/Divisor/Data Type Conversion Inherited'
 * '<S208>' : 'UDC/SlipDetection/E9_5_SlipCtrlCorr/TON/Data Type Conversion Inherited'
 * '<S209>' : 'UDC/SlipDetection/E9_5_SlipCtrlCorr/rateLimit/Saturation Dynamic'
 * '<S210>' : 'UDC/SlipDetection/E9_5_SlipCtrlCorr/rateLimit1/Saturation Dynamic'
 */
#endif                                 /* RTW_HEADER_UDC_h_ */
```

#### UDC_private.h
```c
/********************************************************************
 * COPYRIGHT -- Bernecker + Rainer Industrie-Elektronik Ges.m.b.H.
 ********************************************************************
 * Program: UDC
 * File: UDC_private.h
 * Author: 105055527
 * Created: Thu Mar 02 16:51:06 2017
 ********************************************************************
 * Header for program UDC
 ********************************************************************
 * Generated with B&R Automation Studio Target for Simulink V4.2
 * (ERT based)
 ********************************************************************/

#ifndef RTW_HEADER_UDC_private_h_
#define RTW_HEADER_UDC_private_h_
#include "rtwtypes.h"
#include <bur/plctypes.h>
#ifndef __RTWTYPES_H__
#error This file requires rtwtypes.h to be included
#else
#ifdef TMWTYPES_PREVIOUSLY_INCLUDED
#error This file requires rtwtypes.h to be included before tmwtypes.h
#else

/* Check for inclusion of an incorrect version of rtwtypes.h */
#ifndef RTWTYPES_ID_C08S16I32L32N32F1
#error This code was generated with a different "rtwtypes.h" than the file included
#endif                                 /* RTWTYPES_ID_C08S16I32L32N32F1 */
#endif                                 /* TMWTYPES_PREVIOUSLY_INCLUDED */
#endif                                 /* __RTWTYPES_H__ */

#ifndef MIN
#define MIN(a,b)                       ((a) < (b) ? (a) : (b))
#endif

#ifndef MAX
#define MAX(a,b)                       ((a) > (b) ? (a) : (b))
#endif

void BINARYSEARCH_real32_T(uint32_T *piLeft, uint32_T *piRght, real32_T u, const
  real32_T *pData, uint32_T iHi, struct fUDC* inst);
void LookUp_real32_T_real32_T(real32_T *pY, const real32_T *pYData, real32_T u,
  const real32_T *pUData, uint32_T iHi, struct fUDC* inst);
void BINARYSEARCH_real32_Treal_T(uint32_T *piLeft, uint32_T *piRght, real32_T u,
  const real_T *pData, uint32_T iHi, struct fUDC* inst);
void LookUp_real32_T_real32_Treal_T(real32_T *pY, const real32_T *pYData,
  real32_T u, const real_T *pUData, uint32_T iHi, struct fUDC* inst);
extern uint32_T plook_u32ff_binca(real32_T u, const real32_T bp[], uint32_T
  maxIndex, real32_T *fraction, struct fUDC* inst);
extern real32_T intrp2d_if_u32f_la_pw(const uint32_T bpIndex[], const real32_T
  frac[], const real32_T table[], uint32_T stride, const uint32_T maxIndex[], struct fUDC* inst);
extern uint32_T binsearch_u32f(real32_T u, const real32_T bp[], uint32_T
  startIndex, uint32_T maxIndex, struct fUDC* inst);
extern void UDC_Cell1_Init(rtDW_Cell1_UDC *localDW, struct fUDC* inst);
extern void UDC_Cell1(real32_T rtu_mdotExhWetkgs, real32_T rtu_cpExhJkgK,
                      real32_T rtu_TgSCRInC, real32_T rtu_haWm2K, real32_T
                      rtu_ACatm2, boolean_T rtu_Resetbool, real32_T rtu_I0C,
                      real32_T rtu_TambC, real32_T rtu_mCatkg, real32_T
                      rtu_cCatJkgK, const real32_T rtu_rNH3StorMap_x[5], const
                      real32_T rtu_rNH3StorMap_y[5], rtB_Cell1_UDC *localB,
                      rtDW_Cell1_UDC *localDW, struct fUDC* inst);
extern void UDC_Filter_Init(rtDW_Filter_UDC *localDW, struct fUDC* inst);
extern void UDC_Filter(real32_T rtu_T_filt, boolean_T rtu_reset, real32_T rtu_x0,
  rtB_Filter_UDC *localB, rtDW_Filter_UDC *localDW, struct fUDC* inst);
extern void UDC_TON(boolean_T rtu_IN, real32_T rtu_PT, rtB_TON_UDC *localB,
                    rtDW_TON_UDC *localDW, struct fUDC* inst);
extern void UDC_EnabledSubsystem(boolean_T rtu_0, real32_T rtu_1, real32_T
  *rty_Out1, struct fUDC* inst);
extern void UDC_TP_Init(rtDW_TP_UDC *localDW, struct fUDC* inst);
extern void UDC_TP(boolean_T rtu_IN, real32_T rtu_PT, rtB_TP_UDC *localB,
                   rtDW_TP_UDC *localDW, struct fUDC* inst);
extern void UDC_TOF_Init(rtDW_TOF_UDC *localDW, struct fUDC* inst);
extern void UDC_TOF(boolean_T rtu_IN, real_T rtu_PT, rtB_TOF_UDC *localB,
                    rtDW_TOF_UDC *localDW, struct fUDC* inst);

#endif                                 /* RTW_HEADER_UDC_private_h_ */
```

#### UDC_types.h
```c
/********************************************************************
 * COPYRIGHT -- Bernecker + Rainer Industrie-Elektronik Ges.m.b.H.
 ********************************************************************
 * Program: UDC
 * File: UDC_types.h
 * Author: 105055527
 * Created: Thu Mar 02 16:51:06 2017
 ********************************************************************
 * Header for program UDC
 ********************************************************************
 * Generated with B&R Automation Studio Target for Simulink V4.2
 * (ERT based)
 ********************************************************************/

#ifndef RTW_HEADER_UDC_types_h_
#define RTW_HEADER_UDC_types_h_
#include "rtwtypes.h"
#ifndef MIN
#define MIN(a,b)                       ((a) < (b) ? (a) : (b))
#endif

#ifndef MAX
#define MAX(a,b)                       ((a) > (b) ? (a) : (b))
#endif

/* Forward declaration for rtModel */
typedef struct tag_RTM_UDC RT_MODEL_UDC;

#endif                                 /* RTW_HEADER_UDC_types_h_ */
```

#### rtGetInf.h
```c
/********************************************************************
 * COPYRIGHT -- Bernecker + Rainer Industrie-Elektronik Ges.m.b.H.
 ********************************************************************
 * Program: UDC
 * File: rtGetInf.h
 * Author: 105055527
 * Created: Thu Mar 02 16:51:06 2017
 ********************************************************************
 * Header for program UDC
 ********************************************************************
 * Generated with B&R Automation Studio Target for Simulink V4.2
 * (ERT based)
 ********************************************************************/

#ifndef RTW_HEADER_rtGetInf_h_
#define RTW_HEADER_rtGetInf_h_
#include <stddef.h>
#include "rtwtypes.h"
#include "rt_nonfinite.h"
#ifndef MIN
#define MIN(a,b)                       ((a) < (b) ? (a) : (b))
#endif

#ifndef MAX
#define MAX(a,b)                       ((a) > (b) ? (a) : (b))
#endif

extern real_T rtGetInf(void);
extern real32_T rtGetInfF(void);
extern real_T rtGetMinusInf(void);
extern real32_T rtGetMinusInfF(void);

#endif                                 /* RTW_HEADER_rtGetInf_h_ */
```

#### rtGetNaN.h
```c
/********************************************************************
 * COPYRIGHT -- Bernecker + Rainer Industrie-Elektronik Ges.m.b.H.
 ********************************************************************
 * Program: UDC
 * File: rtGetNaN.h
 * Author: 105055527
 * Created: Thu Mar 02 16:51:06 2017
 ********************************************************************
 * Header for program UDC
 ********************************************************************
 * Generated with B&R Automation Studio Target for Simulink V4.2
 * (ERT based)
 ********************************************************************/

#ifndef RTW_HEADER_rtGetNaN_h_
#define RTW_HEADER_rtGetNaN_h_
#include <stddef.h>
#include "rtwtypes.h"
#include "rt_nonfinite.h"
#ifndef MIN
#define MIN(a,b)                       ((a) < (b) ? (a) : (b))
#endif

#ifndef MAX
#define MAX(a,b)                       ((a) > (b) ? (a) : (b))
#endif

extern real_T rtGetNaN(void);
extern real32_T rtGetNaNF(void);

#endif                                 /* RTW_HEADER_rtGetNaN_h_ */
```

#### rt_nonfinite.h
```c
/********************************************************************
 * COPYRIGHT -- Bernecker + Rainer Industrie-Elektronik Ges.m.b.H.
 ********************************************************************
 * Program: UDC
 * File: rt_nonfinite.h
 * Author: 105055527
 * Created: Thu Mar 02 16:51:06 2017
 ********************************************************************
 * Header for program UDC
 ********************************************************************
 * Generated with B&R Automation Studio Target for Simulink V4.2
 * (ERT based)
 ********************************************************************/

#ifndef RTW_HEADER_rt_nonfinite_h_
#define RTW_HEADER_rt_nonfinite_h_
#include <stddef.h>
#include "rtwtypes.h"
#ifndef MIN
#define MIN(a,b)                       ((a) < (b) ? (a) : (b))
#endif

#ifndef MAX
#define MAX(a,b)                       ((a) > (b) ? (a) : (b))
#endif

extern real_T rtInf;
extern real_T rtMinusInf;
extern real_T rtNaN;
extern real32_T rtInfF;
extern real32_T rtMinusInfF;
extern real32_T rtNaNF;
extern void rt_InitInfAndNaN(size_t realSize);
extern boolean_T rtIsInf(real_T value);
extern boolean_T rtIsInfF(real32_T value);
extern boolean_T rtIsNaN(real_T value);
extern boolean_T rtIsNaNF(real32_T value);
typedef struct {
  struct {
    uint32_T wordH;
    uint32_T wordL;
  } words;
} BigEndianIEEEDouble;

typedef struct {
  struct {
    uint32_T wordL;
    uint32_T wordH;
  } words;
} LittleEndianIEEEDouble;

typedef struct {
  union {
    real32_T wordLreal;
    uint32_T wordLuint;
  } wordL;
} IEEESingle;

#endif                                 /* RTW_HEADER_rt_nonfinite_h_ */
```

#### rtwtypes.h
```c
/********************************************************************
 * COPYRIGHT -- Bernecker + Rainer Industrie-Elektronik Ges.m.b.H.
 ********************************************************************
 * Program: UDC
 * File: rtwtypes.h
 * Author: 105055527
 * Created: Thu Mar 02 16:51:06 2017
 ********************************************************************
 * Header for program UDC
 ********************************************************************
 * Generated with B&R Automation Studio Target for Simulink V4.2
 * (ERT based)
 ********************************************************************/

#ifndef __RTWTYPES_H__
#define __RTWTYPES_H__
#ifndef TRUE
# define TRUE                          (1U)
#endif

#ifndef FALSE
# define FALSE                         (0U)
#endif

#ifndef __TMWTYPES__
#define __TMWTYPES__
#include <limits.h>

/*=======================================================================*
 * Target hardware information
 *   Device type: Intel->x86/Pentium
 *   Number of bits:     char:   8    short:   16    long:  32
 *                       long:  32
 *                       native word size:  32
 *   Byte ordering: LittleEndian
 *   Signed integer division rounds to: Zero
 *   Shift right on a signed integer as arithmetic shift: on
 *=======================================================================*/

/*=======================================================================*
 * Fixed width word size data types:                                     *
 *   int8_T, int16_T, int32_T     - signed 8, 16, or 32 bit integers     *
 *   uint8_T, uint16_T, uint32_T  - unsigned 8, 16, or 32 bit integers   *
 *   real32_T, real64_T           - 32 and 64 bit floating point numbers *
 *=======================================================================*/
typedef signed char int8_T;
typedef unsigned char uint8_T;
typedef short int16_T;
typedef unsigned short uint16_T;
typedef long int32_T;
typedef unsigned long uint32_T;
typedef float real32_T;
typedef double real64_T;

/*===========================================================================*
 * Generic type definitions: real_T, time_T, boolean_T, int_T, uint_T,       *
 *                           ulong_T, char_T and byte_T.                     *
 *===========================================================================*/
typedef double real_T;
typedef double time_T;
typedef unsigned char boolean_T;
typedef long int_T;
typedef unsigned long uint_T;
typedef unsigned long ulong_T;
typedef char char_T;
typedef unsigned char uchar_T;
typedef char_T byte_T;

/*=======================================================================*
 * Min and Max:                                                          *
 *   int8_T, int16_T, int32_T     - signed 8, 16, or 32 bit integers     *
 *   uint8_T, uint16_T, uint32_T  - unsigned 8, 16, or 32 bit integers   *
 *=======================================================================*/
#define MAX_int8_T                     ((int8_T)(127))
#define MIN_int8_T                     ((int8_T)(-128))
#define MAX_uint8_T                    ((uint8_T)(255U))
#define MIN_uint8_T                    ((uint8_T)(0U))
#define MAX_int16_T                    ((int16_T)(32767))
#define MIN_int16_T                    ((int16_T)(-32768))
#define MAX_uint16_T                   ((uint16_T)(65535U))
#define MIN_uint16_T                   ((uint16_T)(0U))
#define MAX_int32_T                    ((int32_T)(2147483647))
#define MIN_int32_T                    ((int32_T)(-2147483647-1))
#define MAX_uint32_T                   ((uint32_T)(0xFFFFFFFFU))
#define MIN_uint32_T                   ((uint32_T)(0U))

/* Logical type definitions */
#if (!defined(__cplusplus)) && (!defined(__true_false_are_keywords))
#  ifndef false
#   define false                       (0U)
#  endif

#  ifndef true
#   define true                        (1U)
#  endif
#endif

/*
 * Simulink Coder assumes the code is compiled on a target using a 2's complement representation
 * for signed integer values.
 */
#if ((SCHAR_MIN + 1) != -SCHAR_MAX)
#error "This code must be compiled using a 2's complement representation for signed integer values"
#endif

/* This ID is used to detect inclusion of an incompatible rtwtypes.h */
#define RTWTYPES_ID_C08S16I32L32N32F1
#else                                  /* __TMWTYPES__ */
#define TMWTYPES_PREVIOUSLY_INCLUDED
#endif                                 /* __TMWTYPES__ */

/* Block D-Work pointer type */
typedef void * pointer_T;

/* Simulink specific types */
#ifndef __SIMSTRUC_TYPES_H__
#define __SIMSTRUC_TYPES_H__

/* Trigger directions: falling, either, and rising */
typedef enum {
  FALLING_ZERO_CROSSING = -1,
  ANY_ZERO_CROSSING = 0,
  RISING_ZERO_CROSSING = 1
} ZCDirection;

/* Previous state of a trigger signal */
typedef uint8_T ZCSigState;

/* Initial value of a trigger zero crossing signal */
#define UNINITIALIZED_ZCSIG            0x03U
#define NEG_ZCSIG                      0x02U
#define POS_ZCSIG                      0x01U
#define ZERO_ZCSIG                     0x00U

/* Current state of a trigger signal */
typedef enum {
  FALLING_ZCEVENT = -1,
  NO_ZCEVENT = 0,
  RISING_ZCEVENT = 1
} ZCEventType;

#endif                                 /* __SIMSTRUC_TYPES_H__ */
#endif                                 /* __RTWTYPES_H__ */

#ifndef MIN
#define MIN(a,b)                       ((a) < (b) ? (a) : (b))
#endif

#ifndef MAX
#define MAX(a,b)                       ((a) > (b) ? (a) : (b))
#endif
```
